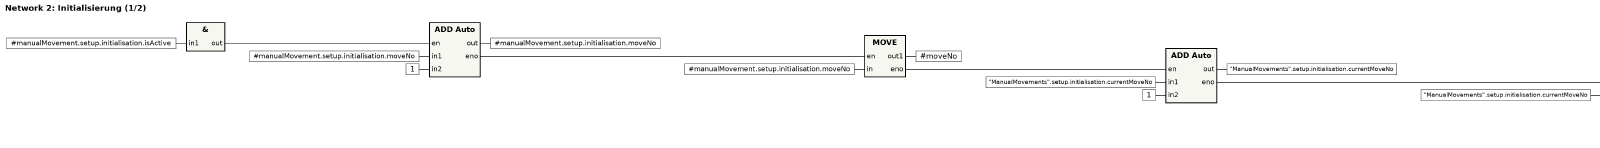
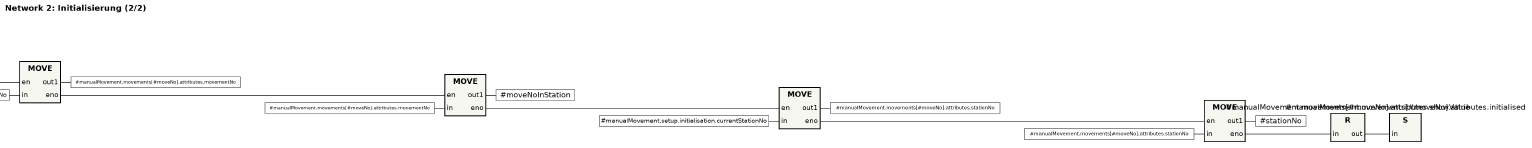
   IF #manualMovement.setup.initialisation.isActive THEN
       #manualMovement.setup.initialisation.moveNo := #manualMovement.setup.initialisation.moveNo + 1;
       #moveNo := #manualMovement.setup.initialisation.moveNo;
       "ManualMovements".setup.initialisation.currentMoveNo := "ManualMovements".setup.initialisation.currentMoveNo + 1;
       #manualMovement.movements[#moveNo].attributes.movementNo := "ManualMovements".setup.initialisation.currentMoveNo;
       #moveNoInStation := #manualMovement.movements[#moveNo].attributes.movementNo;
       #manualMovement.movements[#moveNo].attributes.stationNo := #manualMovement.setup.initialisation.currentStationNo;
       #stationNo := #manualMovement.movements[#moveNo].attributes.stationNo;
       #manualMovement.movements[#moveNo].attributes.showValue := FALSE;
       #manualMovement.movements[#moveNo].attributes.initialised := TRUE;
   END_IF;
END_REGION

REGION Network 3: Initialisierung abgeschlossen?
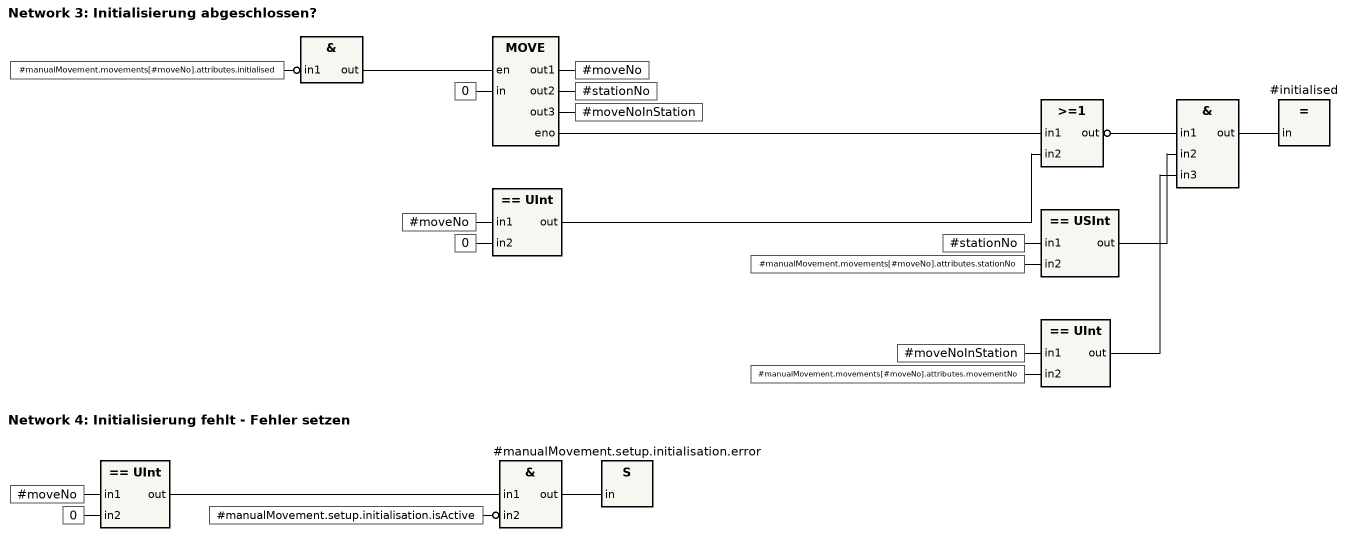
   #_w1 := NOT #manualMovement.movements[#moveNo].attributes.initialised;
   IF #_w1 THEN
       #moveNo := 0;
       #stationNo := 0;
       #moveNoInStation := 0;
   END_IF;
   #initialised := NOT (#_w1 OR (#moveNo = 0)) AND (#stationNo = #manualMovement.movements[#moveNo].attributes.stationNo) AND (#moveNoInStation = #manualMovement.movements[#moveNo].attributes.movementNo);
END_REGION

REGION Network 4: Initialisierung fehlt - Fehler setzen
   IF (#moveNo = 0) AND NOT #manualMovement.setup.initialisation.isActive THEN
       #manualMovement.setup.initialisation.error := TRUE;
   END_IF;
END_REGION

REGION Network 5: Sichtbarkeit
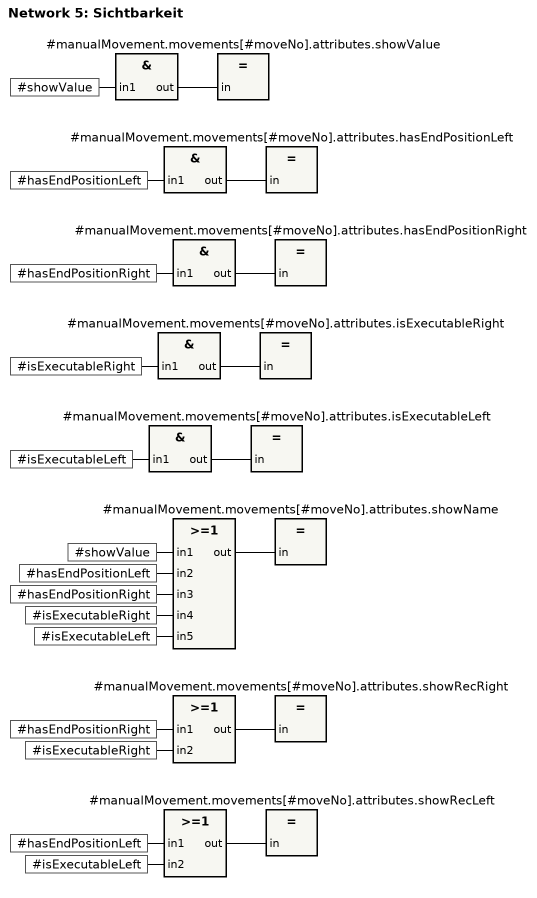
   #manualMovement.movements[#moveNo].attributes.showValue := #showValue;
   #manualMovement.movements[#moveNo].attributes.hasEndPositionLeft := #hasEndPositionLeft;
   #manualMovement.movements[#moveNo].attributes.hasEndPositionRight := #hasEndPositionRight;
   #manualMovement.movements[#moveNo].attributes.isExecutableRight := #isExecutableRight;
   #manualMovement.movements[#moveNo].attributes.isExecutableLeft := #isExecutableLeft;
   #manualMovement.movements[#moveNo].attributes.showName := #showValue OR #hasEndPositionLeft OR #hasEndPositionRight OR #isExecutableRight OR #isExecutableLeft;
   #manualMovement.movements[#moveNo].attributes.showRecRight := #hasEndPositionRight OR #isExecutableRight;
   #manualMovement.movements[#moveNo].attributes.showRecLeft := #hasEndPositionLeft OR #isExecutableLeft;
END_REGION
END_FUNCTION

FUNCTION "InitManualMovements" : Void   // FC909, SCL
{ S7_Optimized_Access := 'TRUE' }
VERSION : 0.1
   VAR_IN_OUT
      movements : Array[0.."SYS_MANUALMOVEMENTS"] of "typeManualMove";
   END_VAR
   VAR_TEMP
      tempCounter : USInt;
   END_VAR
BEGIN
   // Ersteller: Andreas Fast Automation
   // E-Mail: automation@fast-andreas.de
   //
   // Projekt dient zu Demonstrationszwecken und frei genutzt werden.
   //
   // Bausteinbeschreibung:
   // 


   FOR #tempCounter := 0 TO "SYS_MANUALMOVEMENTS" DO
       // Initialise all manual movements
       #movements[#tempCounter].attributes.initialised := false;
       "ManualMovements".movements[#tempCounter].attributes.showValue := false;
       "ManualMovements".movements[#tempCounter].attributes.showName := false;
       "ManualMovements".movements[#tempCounter].attributes.showRecRight := false;
       "ManualMovements".movements[#tempCounter].attributes.showRecLeft := false;
       "ManualMovements".movements[#tempCounter].attributes.isExecutableRight := false;
       "ManualMovements".movements[#tempCounter].attributes.isExecutableLeft := false;
       "ManualMovements".movements[#tempCounter].attributes.hasEndPositionRight := false;
       "ManualMovements".movements[#tempCounter].attributes.hasEndPositionLeft := false;

       #movements[#tempCounter].attributes.stationNo := 0;
       #movements[#tempCounter].attributes.movementNo := 0;
   END_FOR;
END_FUNCTION

// folder: 9. Library/9.2 Actors

FUNCTION_BLOCK "Actor"   // FB9200, FBD
TITLE = Aktoransteuerung
{ S7_Optimized_Access := 'TRUE' }
VERSION : 0.1
// Ersteller: Andreas Fast Automation
// E-Mail: automation@fast-andreas.de
// 
// Projekt dient zu Demonstrationszwecken und frei genutzt werden.
// 
// Bausteinbeschreibung:
// Grundlegende Funktionssteuerung eines Aktors
   VAR_INPUT
      config : USInt;   // Konfiguration Endschalterabfrage (0 = keine, 1 nur GS, 2 = Nur AS, 3 = Beide)
      "one-sided" : Bool;   // Einseitige Ansteuerung (Nur Ansteuerung zur Arbeitsstellung vorhanden, tastend)
      selfLocking : Bool;   // 1 = Selbsthaltung aktiv (Steuerimpuls setzt das Ausgangssignal)
      selfLockingInSetup : Bool;   // 1 = Selbsthaltung nur im Einrichtbetrieb bei einseitiger Spule (Ausgangsansteuerung wird setzend im Einrichten)
      holdEndposition : Bool;   // 1 = hält Ausgangsansteuerung aufrecht, wenn Endposition erreicht wurde
      iniHomePos : Bool;   // Grundstellung erreicht
      iniWorkPos : Bool;   // Arbeitsstellung erreicht
      interlockHome : Bool := true;   // 1 = Ansteuerung Grundstellung freigegeben
      interlockWork : Bool := true;   // 1 = Ansteuerung Arbeitsstellung freigegeben
      reactionTime : Time := t#25ms;   // Endschalter Reaktionsverzögerung
      configNoReleaseCycle : Bool := false;   // 1 = Stationsfreigabe ist zur Ansteuerung nicht notwendig
   END_VAR
   VAR_OUTPUT
      manualMoveNo : UInt;   // Bewegungsnummer für Einrichtfunktion
      homePos : Bool;
      workPos : Bool;
   END_VAR
   VAR_IN_OUT
      actor : "typeActor";
      signals : "typeStationSignals";
      manualMovement : "typeManualMovements";
   END_VAR
   VAR
      statManualHomePos : Bool;
      statManualWorkPos : Bool;
      statSetHomeAct : Bool;
      statSetWorkAct : Bool;
      statActorManualMovement : "ActorManualMovement";
      instReactionHome : TON_TIME;
      instReactionWork : TON_TIME;
   END_VAR
   VAR_TEMP
      tempSelfLocking : Bool;
      tempHomePosConfig : Bool;
      tempWorkPosConfig : Bool;
   END_VAR
BEGIN

REGION Network 1: Selbsthaltung
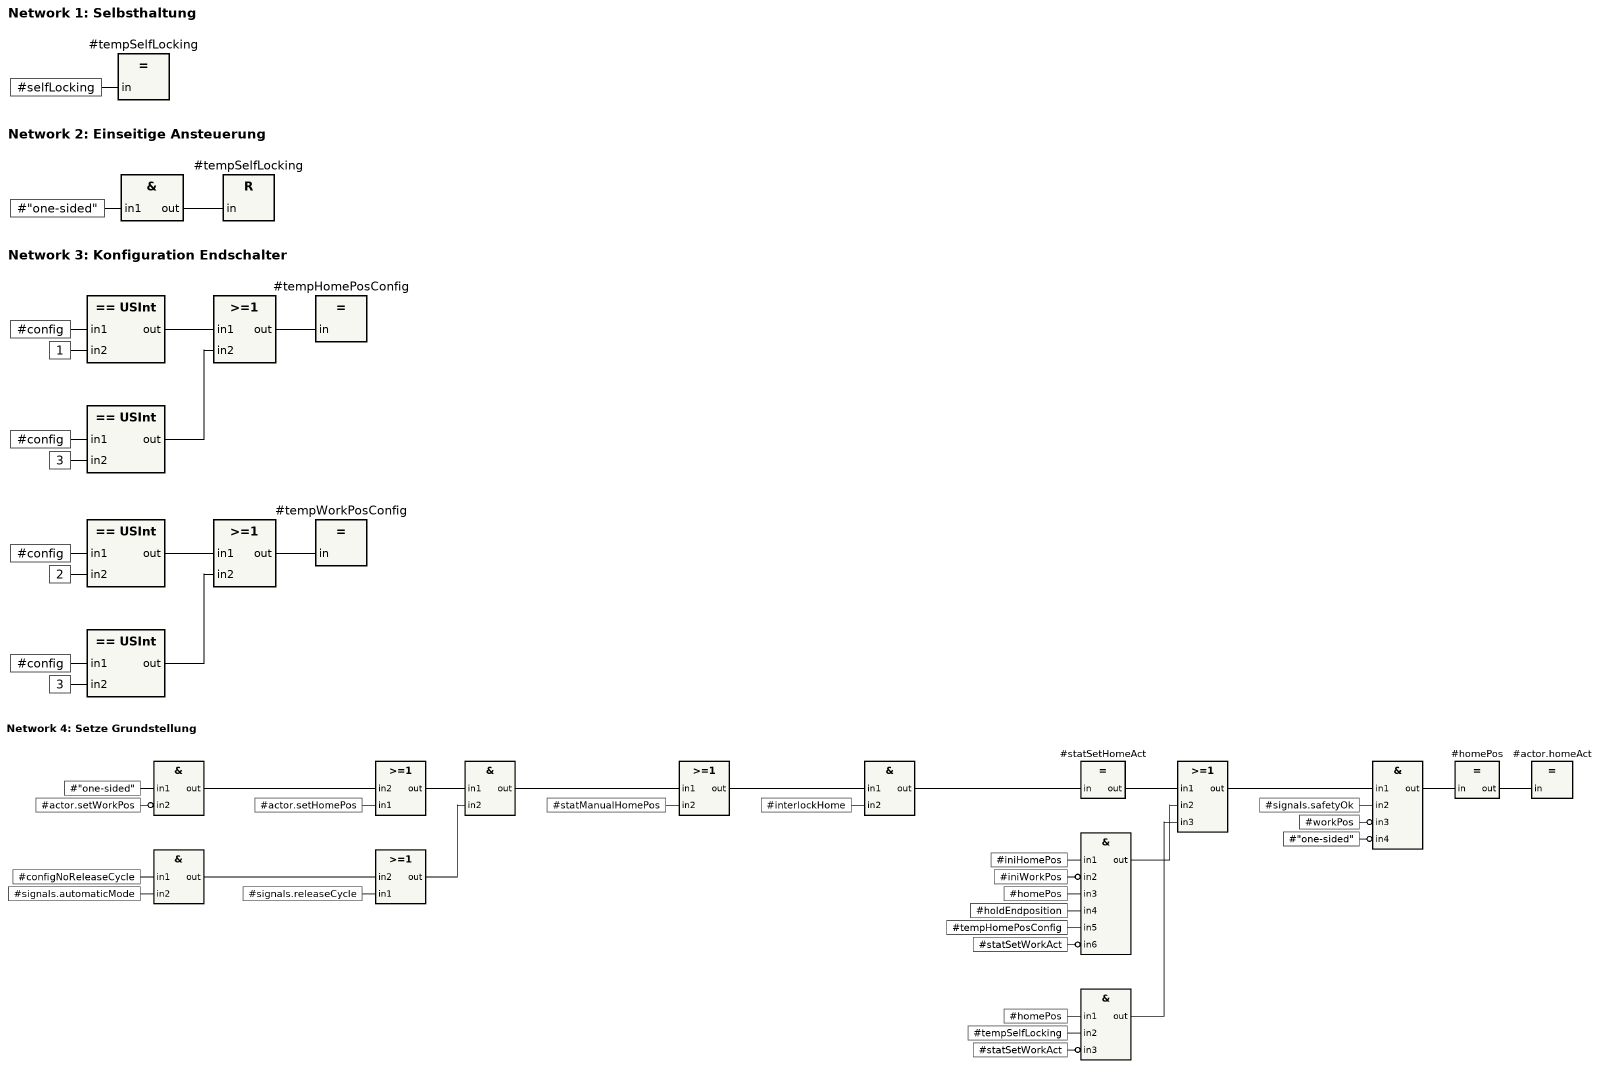
   #tempSelfLocking := #selfLocking;
END_REGION

REGION Network 2: Einseitige Ansteuerung
   IF #"one-sided" THEN #tempSelfLocking := FALSE; END_IF;
END_REGION

REGION Network 3: Konfiguration Endschalter
   // 0 = Ohne Inis
   // 1 = Nur Grundstellungsabfrage
   // 2 = Nur Arbeitstellungsabfrage
   // 3 = Beide Schaltstellungen werden abgefragt
   #tempHomePosConfig := (#config = 1) OR (#config = 3);
   #tempWorkPosConfig := (#config = 2) OR (#config = 3);
END_REGION

REGION Network 4: Setze Grundstellung
   #statSetHomeAct := ((((#"one-sided" AND NOT #actor.setWorkPos) OR #actor.setHomePos) AND ((#configNoReleaseCycle AND #signals.automaticMode) OR #signals.releaseCycle)) OR #statManualHomePos) AND #interlockHome;
   #homePos := (#statSetHomeAct OR (#iniHomePos AND NOT #iniWorkPos AND #homePos AND #holdEndposition AND #tempHomePosConfig AND NOT #statSetWorkAct) OR (#homePos AND #tempSelfLocking AND NOT #statSetWorkAct)) AND #signals.safetyOk AND NOT #workPos AND NOT #"one-sided";
   #actor.homeAct := #homePos;
END_REGION

REGION Network 5: Setze Arbeitsstellung
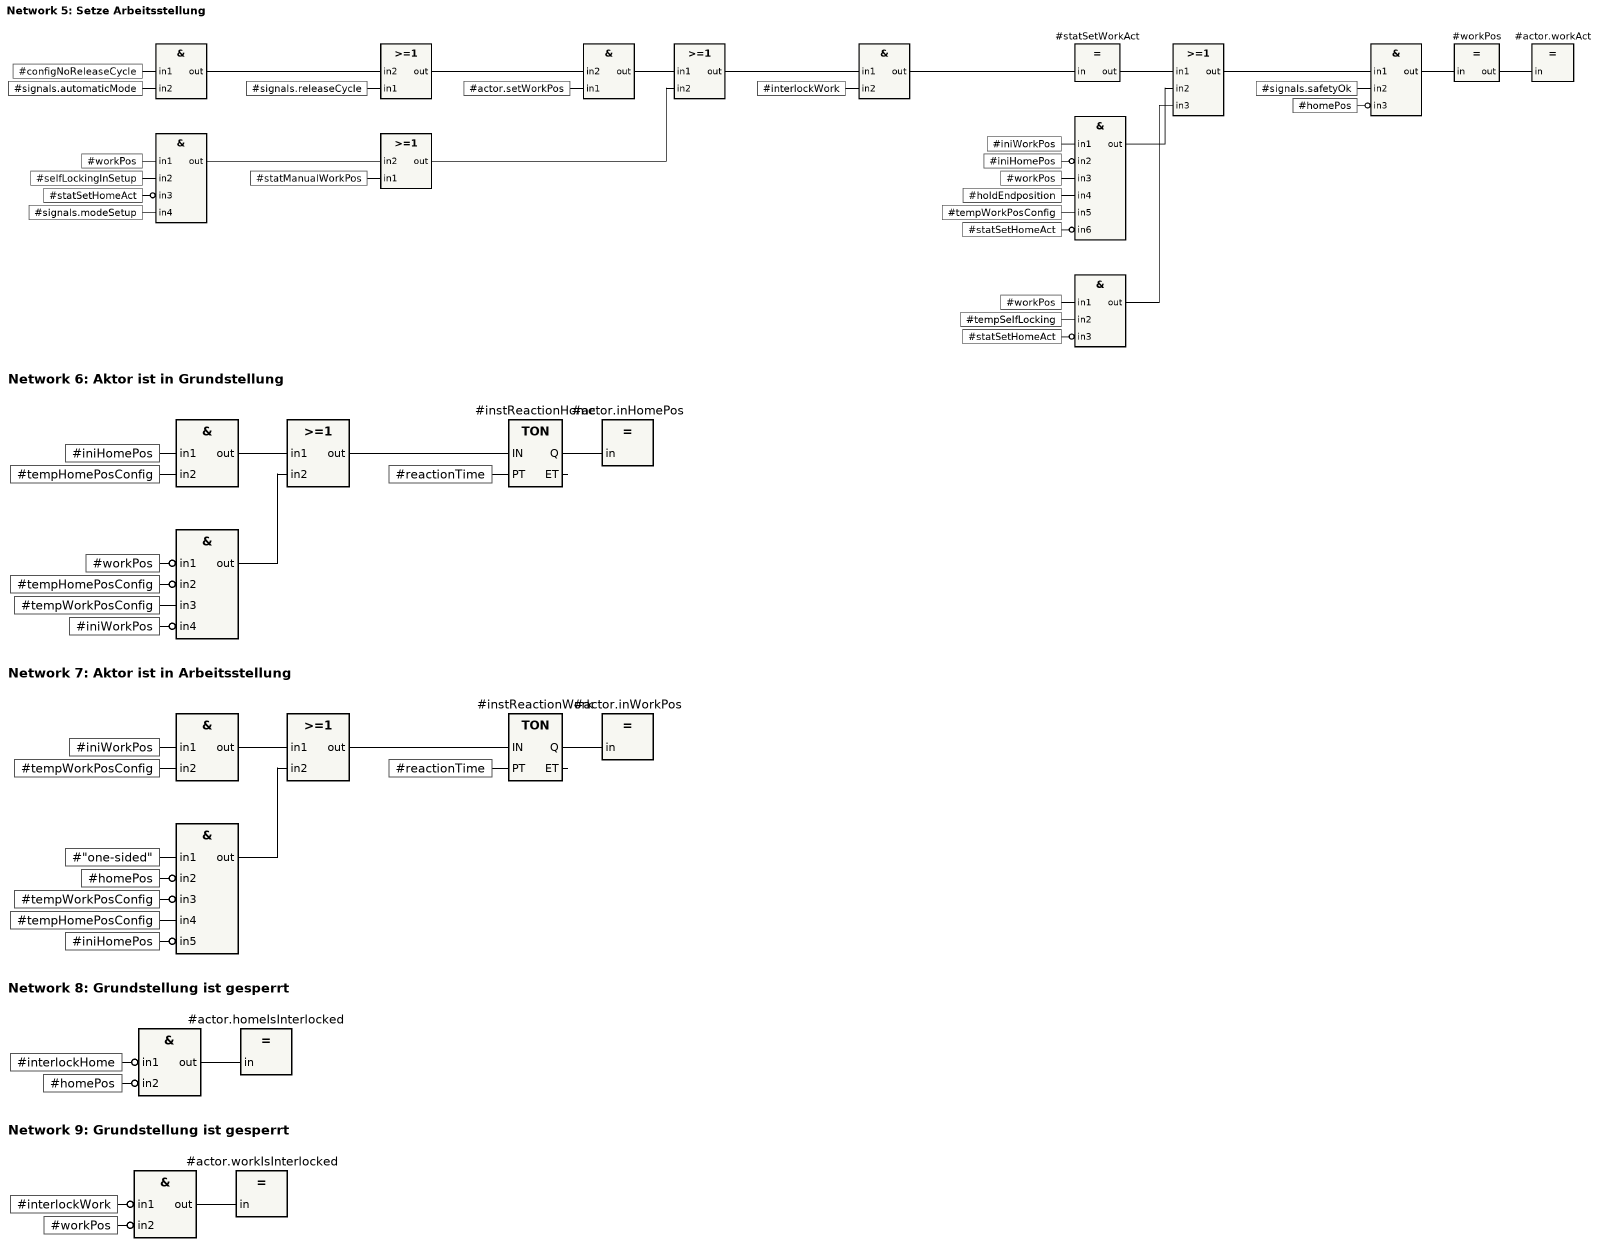
   #statSetWorkAct := ((((#configNoReleaseCycle AND #signals.automaticMode) OR #signals.releaseCycle) AND #actor.setWorkPos) OR (#workPos AND #selfLockingInSetup AND NOT #statSetHomeAct AND #signals.modeSetup) OR #statManualWorkPos) AND #interlockWork;
   #workPos := (#statSetWorkAct OR (#iniWorkPos AND NOT #iniHomePos AND #workPos AND #holdEndposition AND #tempWorkPosConfig AND NOT #statSetHomeAct) OR (#workPos AND #tempSelfLocking AND NOT #statSetHomeAct)) AND #signals.safetyOk AND NOT #homePos;
   #actor.workAct := #workPos;
END_REGION

REGION Network 6: Aktor ist in Grundstellung
   #instReactionHome(IN := (#iniHomePos AND #tempHomePosConfig) OR (NOT #workPos AND NOT #tempHomePosConfig AND #tempWorkPosConfig AND NOT #iniWorkPos),   // TON
                     PT := #reactionTime);
   #actor.inHomePos := #instReactionHome.Q;
END_REGION

REGION Network 7: Aktor ist in Arbeitsstellung
   #instReactionWork(IN := (#iniWorkPos AND #tempWorkPosConfig) OR (#"one-sided" AND NOT #homePos AND NOT #tempWorkPosConfig AND #tempHomePosConfig AND NOT #iniHomePos),   // TON
                     PT := #reactionTime);
   #actor.inWorkPos := #instReactionWork.Q;
END_REGION

REGION Network 8: Grundstellung ist gesperrt
   #actor.homeIsInterlocked := NOT #interlockHome AND NOT #homePos;
END_REGION

REGION Network 9: Grundstellung ist gesperrt
   #actor.workIsInterlocked := NOT #interlockWork AND NOT #workPos;
END_REGION

REGION Network 10: Steuerung Einrichtbewegung eines Aktors
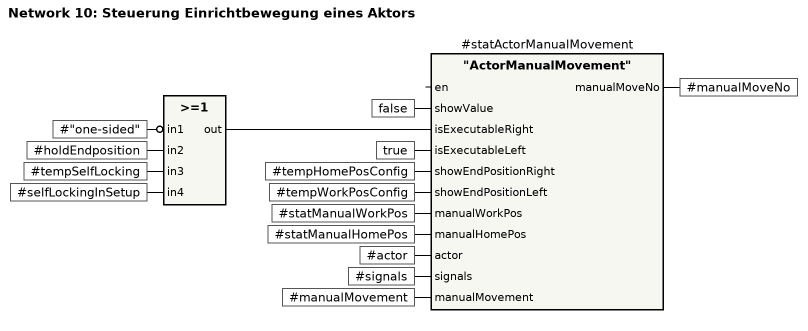
   #statActorManualMovement(showValue := false,   // "ActorManualMovement"
                           isExecutableRight := NOT #"one-sided" OR #holdEndposition OR #tempSelfLocking OR #selfLockingInSetup,
                           isExecutableLeft := true,
                           showEndPositionRight := #tempHomePosConfig,
                           showEndPositionLeft := #tempWorkPosConfig,
                           manualWorkPos := #statManualWorkPos,
                           manualHomePos := #statManualHomePos,
                           actor := #actor,
                           signals := #signals,
                           manualMovement := #manualMovement,
                           manualMoveNo => #manualMoveNo);
END_REGION
END_FUNCTION_BLOCK

FUNCTION_BLOCK "Actor_Reserved"   // FB9201, FBD
TITLE = Aktor als reservierter Platzhalter
{ S7_Optimized_Access := 'TRUE' }
VERSION : 0.1
// Ersteller: Andreas Fast Automation
// E-Mail: automation@fast-andreas.de
// 
// Projekt dient zu Demonstrationszwecken und frei genutzt werden.
// 
// Bausteinbeschreibung:
   VAR_OUTPUT
      manualMoveNo : UInt;   // Bewegungsnummer für Einrichtfunktion
   END_VAR
   VAR_IN_OUT
      manualMovement : "typeManualMovements";
   END_VAR
   VAR
      statActorManualMovement : "ActorManualMovement";
      sudtActor : "typeActor";
      sudtSignals : "typeStationSignals";
   END_VAR
BEGIN

REGION Network 1: Steuerung Einrichtbewegung eines Aktors
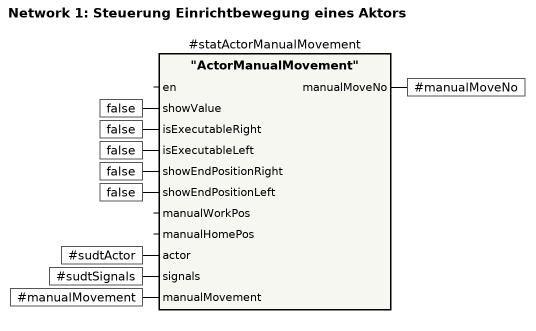
   #statActorManualMovement(showValue := false,   // "ActorManualMovement"
                           isExecutableRight := false,
                           isExecutableLeft := false,
                           showEndPositionRight := false,
                           showEndPositionLeft := false,
                           actor := #sudtActor,
                           signals := #sudtSignals,
                           manualMovement := #manualMovement,
                           manualMoveNo => #manualMoveNo);
END_REGION
END_FUNCTION_BLOCK

// folder: 9. Library/9.2 Actors/9.2.1 Cylinders

FUNCTION_BLOCK "Cylinder_2Out2In"   // FB9211, FBD
TITLE = Valve 2 Outs/2Ins
{ S7_Optimized_Access := 'TRUE' }
VERSION : 0.1
// Ersteller: Andreas Fast Automation
// E-Mail: automation@fast-andreas.de
// 
// Projekt dient zu Demonstrationszwecken und frei genutzt werden.
// 
// Bausteinbeschreibung:
// Ventilansteuerung
// Ansteuerung wird in AS/GS gehalten wenn zugehörige Endstellung vorhanden ist, selbst wenn die Aktoransteuerung rückgesetzt wird.
   VAR_INPUT
      iniHomePos : Bool;   // Grundstellung erreicht
      iniWorkPos : Bool;   // Arbeitsstellung erreicht
      interlockHome : Bool := true;   // 1 = Ansteuerung Grundstellung freigegeben
      interlockWork : Bool := true;   // 1 = Ansteuerung Arbeitsstellung freigegeben
      reactionTime : Time := t#25ms;   // Endschalter Reaktionsverzögerung
      monitoringTime : Time := T#10s;   // Überwachungszeit für Laufzeitfehler
      holdEndposition : Bool := true;   // 1 = hält Ausgangsansteuerung aufrecht, wenn Endposition erreicht wurde
   END_VAR
   VAR_OUTPUT
      manualMoveNo : UInt;   // Bewegungsnummer für Einrichtfunktion
      homePos : Bool;
      workPos : Bool;
   END_VAR
   VAR_IN_OUT
      actor : "typeActor_2Out2In";
      signals : "typeStationSignals";
      manualMovement : "typeManualMovements";
   END_VAR
   VAR
      instActor : "Actor";
      statActor : "typeActor";
      instMonitoringHome : TON_TIME;
      instMonitoringWork : TON_TIME;
   END_VAR
BEGIN

REGION Network 1: Verbinde Aktorsignale vor Aktoransteuerung
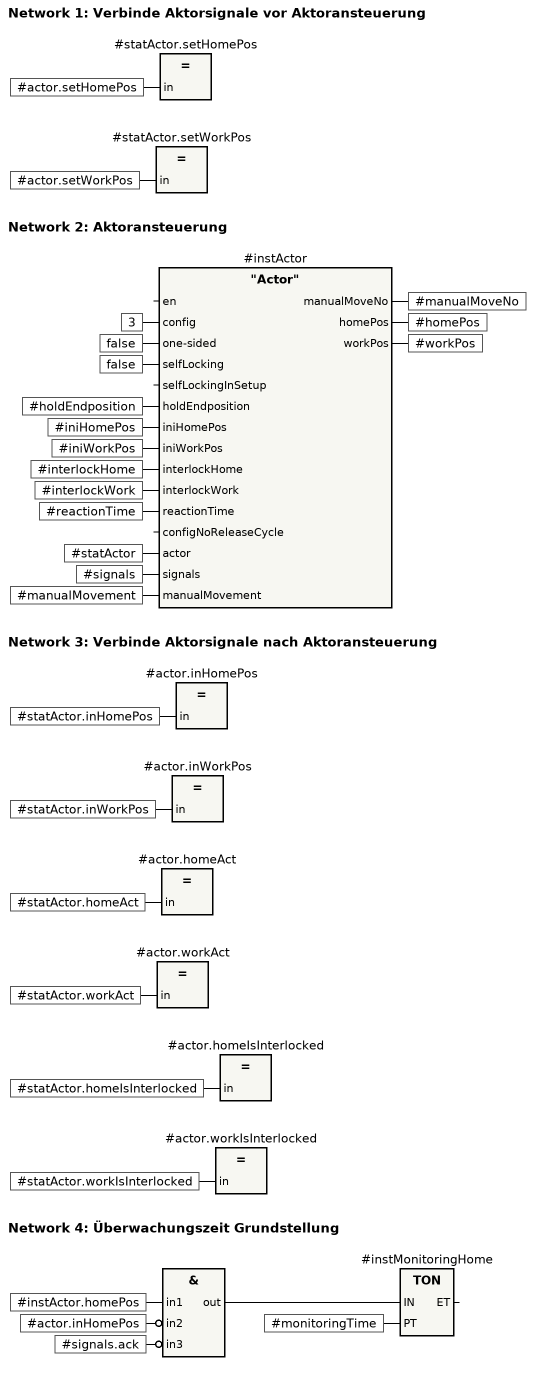
   #statActor.setHomePos := #actor.setHomePos;
   #statActor.setWorkPos := #actor.setWorkPos;
END_REGION

REGION Network 2: Aktoransteuerung
   #instActor(config := 3,   // "Actor"
              "one-sided" := false,
              selfLocking := false,
              holdEndposition := #holdEndposition,
              iniHomePos := #iniHomePos,
              iniWorkPos := #iniWorkPos,
              interlockHome := #interlockHome,
              interlockWork := #interlockWork,
              reactionTime := #reactionTime,
              actor := #statActor,
              signals := #signals,
              manualMovement := #manualMovement,
              manualMoveNo => #manualMoveNo,
              homePos => #homePos,
              workPos => #workPos);
END_REGION

REGION Network 3: Verbinde Aktorsignale nach Aktoransteuerung
   #actor.inHomePos := #statActor.inHomePos;
   #actor.inWorkPos := #statActor.inWorkPos;
   #actor.homeAct := #statActor.homeAct;
   #actor.workAct := #statActor.workAct;
   #actor.homeIsInterlocked := #statActor.homeIsInterlocked;
   #actor.workIsInterlocked := #statActor.workIsInterlocked;
END_REGION

REGION Network 4: Überwachungszeit Grundstellung
   #instMonitoringHome(IN := #instActor.homePos AND NOT #actor.inHomePos AND NOT #signals.ack,   // TON
                       PT := #monitoringTime);
END_REGION

REGION Network 5: Überwachungszeit Arbeitsstellung
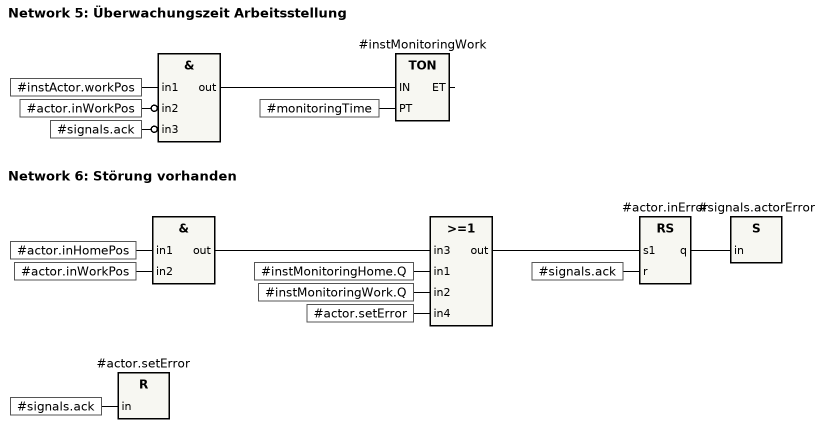
   #instMonitoringWork(IN := #instActor.workPos AND NOT #actor.inWorkPos AND NOT #signals.ack,   // TON
                       PT := #monitoringTime);
END_REGION

REGION Network 6: Störung vorhanden
   IF #signals.ack THEN
       #actor.inError := FALSE;   // RS flip-flop
   END_IF;
   IF (#actor.inHomePos AND #actor.inWorkPos) OR #instMonitoringHome.Q OR #instMonitoringWork.Q OR #actor.setError THEN
       #actor.inError := TRUE;
   END_IF;
   IF #actor.inError THEN #signals.actorError := TRUE; END_IF;
   IF #signals.ack THEN #actor.setError := FALSE; END_IF;
END_REGION
END_FUNCTION_BLOCK

FUNCTION_BLOCK "Cylinder_1Out2In"   // FB9212, FBD
TITLE = Valve 1 Outs/2Ins
{ S7_Optimized_Access := 'TRUE' }
VERSION : 0.1
// Ersteller: Andreas Fast Automation
// E-Mail: automation@fast-andreas.de
// 
// Projekt dient zu Demonstrationszwecken und frei genutzt werden.
// 
// Bausteinbeschreibung:
// Ventilansteuerung
// Ansteuerung wird in AS/GS gehalten wenn zugehörige Endstellung vorhanden ist, selbst wenn die Aktoransteuerung rückgesetzt wird.
   VAR_INPUT
      iniHomePos : Bool;   // Grundstellung erreicht
      iniWorkPos : Bool;   // Arbeitsstellung erreicht
      interlockWork : Bool := true;   // 1 = Ansteuerung Arbeitsstellung freigegeben
      reactionTime : Time := t#25ms;   // Endschalter Reaktionsverzögerung
      monitoringTime : Time := T#10s;   // Überwachungszeit für Laufzeitfehler
      holdEndposition : Bool := false;   // 1 = hält Ausgangsansteuerung aufrecht, wenn Endposition erreicht wurde
   END_VAR
   VAR_OUTPUT
      manualMoveNo : UInt;   // Bewegungsnummer für Einrichtfunktion
      workPos : Bool;   // SPS-Ausgang Ansteuerung Arbeitsstellung
   END_VAR
   VAR_IN_OUT
      actor : "typeActor_1Out2In";
      signals : "typeStationSignals";
      manualMovement : "typeManualMovements";
   END_VAR
   VAR
      instActor : "Actor";
      statActor : "typeActor";
      instMonitoringHome : TON_TIME;
      instMonitoringWork : TON_TIME;
   END_VAR
BEGIN

REGION Network 1: Verbinde Aktorsignale vor Aktoransteuerung
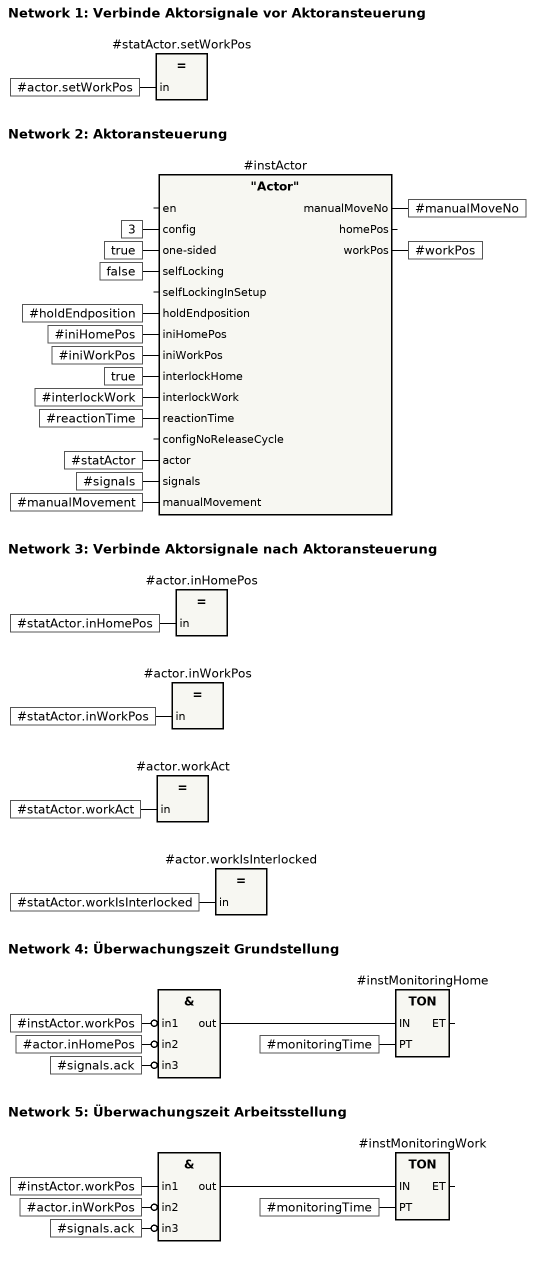
   #statActor.setWorkPos := #actor.setWorkPos;
END_REGION

REGION Network 2: Aktoransteuerung
   #instActor(config := 3,   // "Actor"
              "one-sided" := true,
              selfLocking := false,
              holdEndposition := #holdEndposition,
              iniHomePos := #iniHomePos,
              iniWorkPos := #iniWorkPos,
              interlockHome := true,
              interlockWork := #interlockWork,
              reactionTime := #reactionTime,
              actor := #statActor,
              signals := #signals,
              manualMovement := #manualMovement,
              manualMoveNo => #manualMoveNo,
              workPos => #workPos);
END_REGION

REGION Network 3: Verbinde Aktorsignale nach Aktoransteuerung
   #actor.inHomePos := #statActor.inHomePos;
   #actor.inWorkPos := #statActor.inWorkPos;
   #actor.workAct := #statActor.workAct;
   #actor.workIsInterlocked := #statActor.workIsInterlocked;
END_REGION

REGION Network 4: Überwachungszeit Grundstellung
   #instMonitoringHome(IN := NOT #instActor.workPos AND NOT #actor.inHomePos AND NOT #signals.ack,   // TON
                       PT := #monitoringTime);
END_REGION

REGION Network 5: Überwachungszeit Arbeitsstellung
   #instMonitoringWork(IN := #instActor.workPos AND NOT #actor.inWorkPos AND NOT #signals.ack,   // TON
                       PT := #monitoringTime);
END_REGION

REGION Network 6: Störung vorhanden
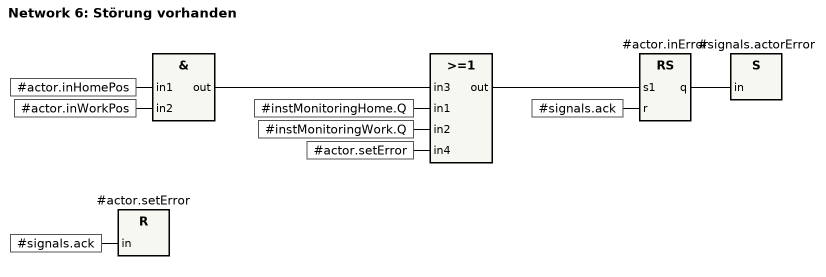
   IF #signals.ack THEN
       #actor.inError := FALSE;   // RS flip-flop
   END_IF;
   IF (#actor.inHomePos AND #actor.inWorkPos) OR #instMonitoringHome.Q OR #instMonitoringWork.Q OR #actor.setError THEN
       #actor.inError := TRUE;
   END_IF;
   IF #actor.inError THEN #signals.actorError := TRUE; END_IF;
   IF #signals.ack THEN #actor.setError := FALSE; END_IF;
END_REGION
END_FUNCTION_BLOCK

FUNCTION_BLOCK "Cylinder_2Out0In (ungetestet)"   // FB9213, FBD
TITLE = Valve 2 Outs/0Ins
{ S7_Optimized_Access := 'TRUE' }
VERSION : 0.1
// Ersteller: Andreas Fast Automation
// E-Mail: automation@fast-andreas.de
// 
// Projekt dient zu Demonstrationszwecken und frei genutzt werden.
// 
// Bausteinbeschreibung:
// Ventilansteuerung
// Ansteuerung wird in AS/GS gehalten wenn zugehörige Endstellung vorhanden ist, selbst wenn die Aktoransteuerung rückgesetzt wird.
   VAR_INPUT
      interlockHome : Bool := true;   // 1 = Ansteuerung Grundstellung freigegeben
      interlockWork : Bool := true;   // 1 = Ansteuerung Arbeitsstellung freigegeben
      reactionTime : Time := t#25ms;   // Endschalter Reaktionsverzögerung
   END_VAR
   VAR_OUTPUT
      manualMoveNo : UInt;   // Bewegungsnummer für Einrichtfunktion
      homePos : Bool;
      workPos : Bool;
   END_VAR
   VAR_IN_OUT
      actor : "typeActor_2Out0In";
      signals : "typeStationSignals";
      manualMovement : "typeManualMovements";
   END_VAR
   VAR
      instActor : "Actor";
      statActor : "typeActor";
   END_VAR
BEGIN

REGION Network 1: Verbinde Aktorsignale vor Aktoransteuerung
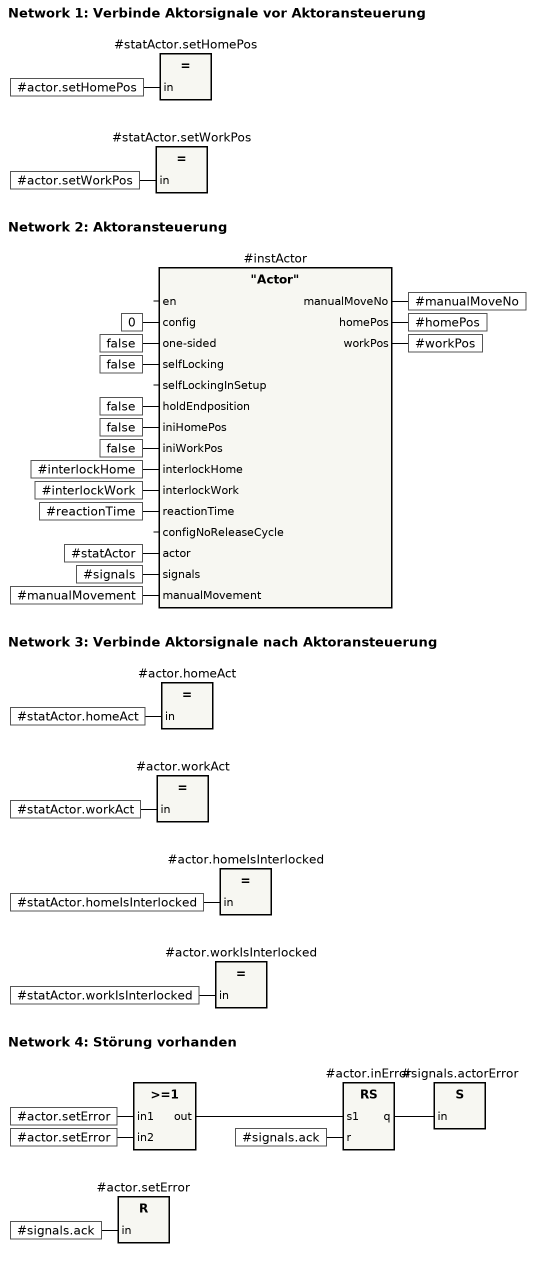
   #statActor.setHomePos := #actor.setHomePos;
   #statActor.setWorkPos := #actor.setWorkPos;
END_REGION

REGION Network 2: Aktoransteuerung
   #instActor(config := 0,   // "Actor"
              "one-sided" := false,
              selfLocking := false,
              holdEndposition := false,
              iniHomePos := false,
              iniWorkPos := false,
              interlockHome := #interlockHome,
              interlockWork := #interlockWork,
              reactionTime := #reactionTime,
              actor := #statActor,
              signals := #signals,
              manualMovement := #manualMovement,
              manualMoveNo => #manualMoveNo,
              homePos => #homePos,
              workPos => #workPos);
END_REGION

REGION Network 3: Verbinde Aktorsignale nach Aktoransteuerung
   #actor.homeAct := #statActor.homeAct;
   #actor.workAct := #statActor.workAct;
   #actor.homeIsInterlocked := #statActor.homeIsInterlocked;
   #actor.workIsInterlocked := #statActor.workIsInterlocked;
END_REGION

REGION Network 4: Störung vorhanden
   IF #signals.ack THEN
       #actor.inError := FALSE;   // RS flip-flop
   END_IF;
   IF #actor.setError OR #actor.setError THEN #actor.inError := TRUE; END_IF;
   IF #actor.inError THEN #signals.actorError := TRUE; END_IF;
   IF #signals.ack THEN #actor.setError := FALSE; END_IF;
END_REGION
END_FUNCTION_BLOCK

FUNCTION_BLOCK "Cylinder_2Out1In (ungetestet)"   // FB9214, FBD
TITLE = Valve 2 Outs/1Ins
{ S7_Optimized_Access := 'TRUE' }
VERSION : 0.1
// Ersteller: Andreas Fast Automation
// E-Mail: automation@fast-andreas.de
// 
// Projekt dient zu Demonstrationszwecken und frei genutzt werden.
// 
// Bausteinbeschreibung:
// Ventilansteuerung
// Ansteuerung wird in AS/GS gehalten wenn zugehörige Endstellung vorhanden ist, selbst wenn die Aktoransteuerung rückgesetzt wird.
   VAR_INPUT
      config : Bool;   // 0 = Ini zeigt Grundstellung erreicht / 1 = Ini zeigt Arbeitsstellung erreicht
      iniEndPos : Bool;   // SPS-Eingang Endposition erreicht
      interlockHome : Bool := true;   // 1 = Ansteuerung Grundstellung freigegeben
      interlockWork : Bool := true;   // 1 = Ansteuerung Arbeitsstellung freigegeben
      reactionTime : Time := t#25ms;   // Endschalter Reaktionsverzögerung
      monitoringTime : Time := T#10s;   // Überwachungszeit für Laufzeitfehler
      holdEndposition : Bool := false;   // 1 = hält Ausgangsansteuerung aufrecht, wenn Endposition erreicht wurde
   END_VAR
   VAR_OUTPUT
      manualMoveNo : UInt;   // Bewegungsnummer für Einrichtfunktion
      homePos : Bool;   // SPS-Ausgang Ansteuerung Grundstellung
      workPos : Bool;   // SPS-Ausgang Ansteuerung Arbeitsstellung
   END_VAR
   VAR_IN_OUT
      actor : "typeActor_2Out1In";
      signals : "typeStationSignals";
      manualMovement : "typeManualMovements";
   END_VAR
   VAR
      instActor : "Actor";
      statActor : "typeActor";
      instMonitoringHome : TON_TIME;
      instMonitoringWork : TON_TIME;
   END_VAR
   VAR_TEMP
      tusiConfig : USInt;
      txInHomePos : Bool;
      txInWorkPos : Bool;
   END_VAR
BEGIN

REGION Network 1: Verbinde Aktorsignale vor Aktoransteuerung
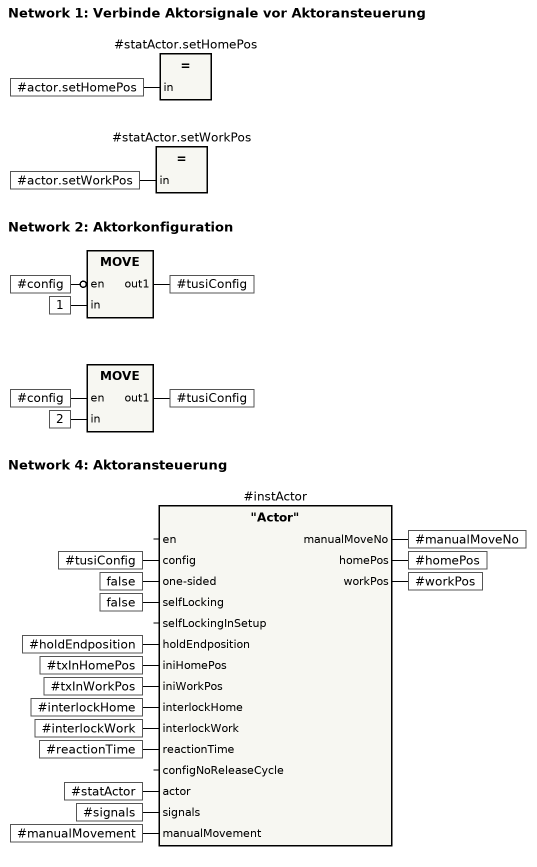
   #statActor.setHomePos := #actor.setHomePos;
   #statActor.setWorkPos := #actor.setWorkPos;
END_REGION

REGION Network 2: Aktorkonfiguration
   IF NOT #config THEN #tusiConfig := 1; END_IF;
   IF #config THEN #tusiConfig := 2; END_IF;
END_REGION

REGION Network 3 (SCL): Endschalter in Grundstellung/Arbeitsstellung

   IF NOT #config THEN // if sensor is checking home position
       #txInHomePos := #iniEndPos;
       #txInWorkPos := NOT #iniEndPos;

   ELSE // sensor is checking work position
       #txInWorkPos := #iniEndPos;
       #txInHomePos := NOT #iniEndPos;
   END_IF;
END_REGION

REGION Network 4: Aktoransteuerung
   #instActor(config := #tusiConfig,   // "Actor"
              "one-sided" := false,
              selfLocking := false,
              holdEndposition := #holdEndposition,
              iniHomePos := #txInHomePos,
              iniWorkPos := #txInWorkPos,
              interlockHome := #interlockHome,
              interlockWork := #interlockWork,
              reactionTime := #reactionTime,
              actor := #statActor,
              signals := #signals,
              manualMovement := #manualMovement,
              manualMoveNo => #manualMoveNo,
              homePos => #homePos,
              workPos => #workPos);
END_REGION

REGION Network 5: Verbinde Aktorsignale nach Aktoransteuerung
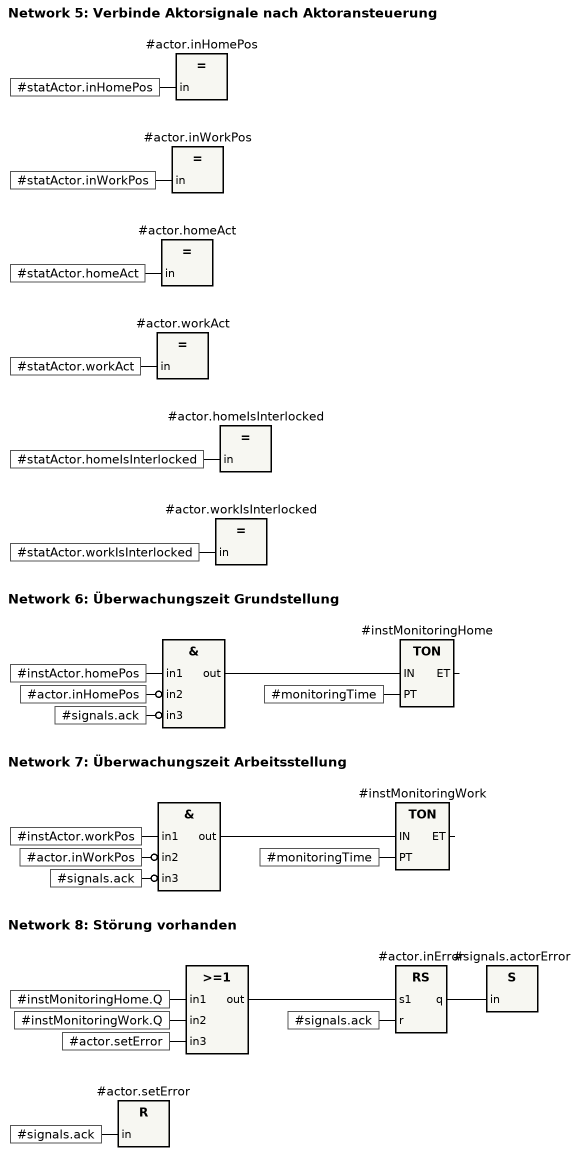
   #actor.inHomePos := #statActor.inHomePos;
   #actor.inWorkPos := #statActor.inWorkPos;
   #actor.homeAct := #statActor.homeAct;
   #actor.workAct := #statActor.workAct;
   #actor.homeIsInterlocked := #statActor.homeIsInterlocked;
   #actor.workIsInterlocked := #statActor.workIsInterlocked;
END_REGION

REGION Network 6: Überwachungszeit Grundstellung
   #instMonitoringHome(IN := #instActor.homePos AND NOT #actor.inHomePos AND NOT #signals.ack,   // TON
                       PT := #monitoringTime);
END_REGION

REGION Network 7: Überwachungszeit Arbeitsstellung
   #instMonitoringWork(IN := #instActor.workPos AND NOT #actor.inWorkPos AND NOT #signals.ack,   // TON
                       PT := #monitoringTime);
END_REGION

REGION Network 8: Störung vorhanden
   IF #signals.ack THEN
       #actor.inError := FALSE;   // RS flip-flop
   END_IF;
   IF #instMonitoringHome.Q OR #instMonitoringWork.Q OR #actor.setError THEN #actor.inError := TRUE; END_IF;
   IF #actor.inError THEN #signals.actorError := TRUE; END_IF;
   IF #signals.ack THEN #actor.setError := FALSE; END_IF;
END_REGION
END_FUNCTION_BLOCK

FUNCTION_BLOCK "Cylinder_1Out1In (ungetestet)"   // FB9215, FBD
TITLE = Valve 1 Out/1In
{ S7_Optimized_Access := 'TRUE' }
VERSION : 0.1
// Ersteller: Andreas Fast Automation
// E-Mail: automation@fast-andreas.de
// 
// Projekt dient zu Demonstrationszwecken und frei genutzt werden.
// 
// Bausteinbeschreibung:
// Ventilansteuerung
// Ansteuerung wird in AS/GS gehalten wenn zugehörige Endstellung vorhanden ist, selbst wenn die Aktoransteuerung rückgesetzt wird.
   VAR_INPUT
      config : Bool;   // 0 = Ini zeigt Grundstellung erreicht / 1 = Ini zeigt Arbeitsstellung erreicht
      iniEndPos : Bool;   // SPS-Eingang Endposition erreicht
      interlockWork : Bool := true;   // 1 = Ansteuerung Arbeitsstellung freigegeben
      reactionTime : Time := t#25ms;   // Endschalter Reaktionsverzögerung
      monitoringTime : Time := T#10s;   // Überwachungszeit für Laufzeitfehler
      holdEndposition : Bool := false;   // 1 = hält Ausgangsansteuerung aufrecht, wenn Endposition erreicht wurde
      selfLockingInSetup : Bool;   // 1 = Selbsthaltung nur im Einrichtbetrieb (zweiseitige Ausgangsansteuerung setzend)
   END_VAR
   VAR_OUTPUT
      manualMoveNo : UInt;   // Bewegungsnummer für Einrichtfunktion
      workPos : Bool;   // SPS-Ausgang Ansteuerung Arbeitsstellung
   END_VAR
   VAR_IN_OUT
      actor : "typeActor_1Out1In";
      signals : "typeStationSignals";
      manualMovement : "typeManualMovements";
   END_VAR
   VAR
      instActor : "Actor";
      statActor : "typeActor";
      instMonitoringHome : TON_TIME;
      instMonitoringWork : TON_TIME;
   END_VAR
   VAR_TEMP
      tusiConfig : USInt;
      txInHomePos : Bool;
      txInWorkPos : Bool;
      txsetzendimeinrichten : Bool;
   END_VAR
BEGIN

REGION Network 1: Verbinde Aktorsignale vor Aktoransteuerung
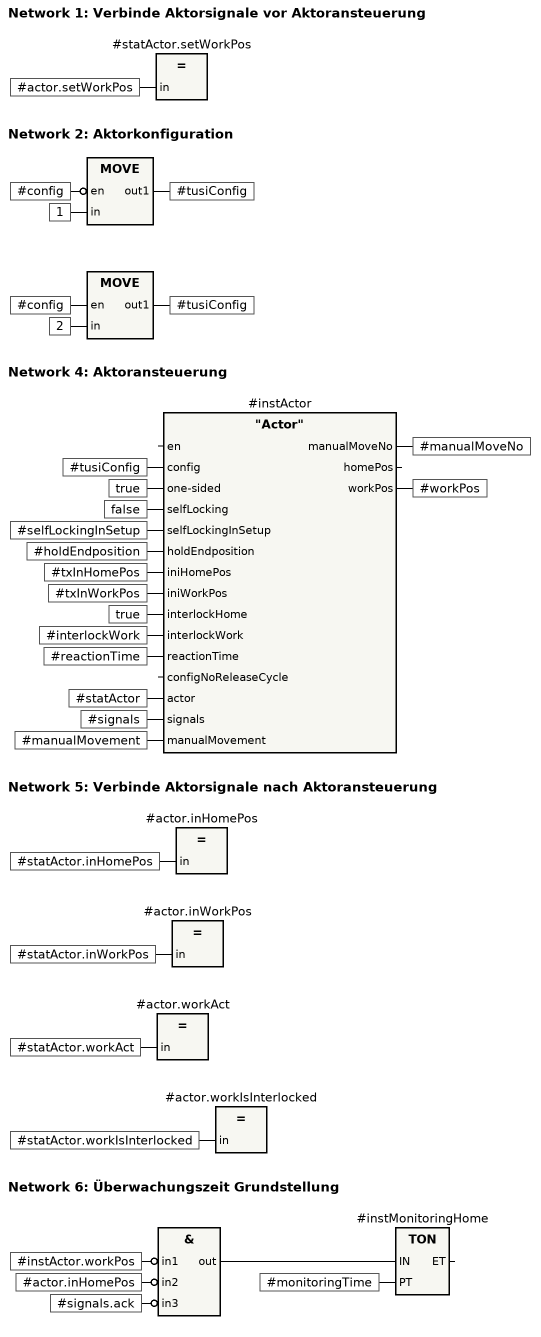
   #statActor.setWorkPos := #actor.setWorkPos;
END_REGION

REGION Network 2: Aktorkonfiguration
   IF NOT #config THEN #tusiConfig := 1; END_IF;
   IF #config THEN #tusiConfig := 2; END_IF;
END_REGION

REGION Network 3 (SCL): Endschalter in Grundstellung/Arbeitsstellung

   IF NOT #config THEN // if sensor is checking home position
       #txInHomePos := #iniEndPos;
       #txInWorkPos := NOT #iniEndPos;

   ELSE // sensor is checking work position
       #txInWorkPos := #iniEndPos;
       #txInHomePos := NOT #iniEndPos;
   END_IF;
END_REGION

REGION Network 4: Aktoransteuerung
   #instActor(config := #tusiConfig,   // "Actor"
              "one-sided" := true,
              selfLocking := false,
              selfLockingInSetup := #selfLockingInSetup,
              holdEndposition := #holdEndposition,
              iniHomePos := #txInHomePos,
              iniWorkPos := #txInWorkPos,
              interlockHome := true,
              interlockWork := #interlockWork,
              reactionTime := #reactionTime,
              actor := #statActor,
              signals := #signals,
              manualMovement := #manualMovement,
              manualMoveNo => #manualMoveNo,
              workPos => #workPos);
END_REGION

REGION Network 5: Verbinde Aktorsignale nach Aktoransteuerung
   #actor.inHomePos := #statActor.inHomePos;
   #actor.inWorkPos := #statActor.inWorkPos;
   #actor.workAct := #statActor.workAct;
   #actor.workIsInterlocked := #statActor.workIsInterlocked;
END_REGION

REGION Network 6: Überwachungszeit Grundstellung
   #instMonitoringHome(IN := NOT #instActor.workPos AND NOT #actor.inHomePos AND NOT #signals.ack,   // TON
                       PT := #monitoringTime);
END_REGION

REGION Network 7: Überwachungszeit Arbeitsstellung
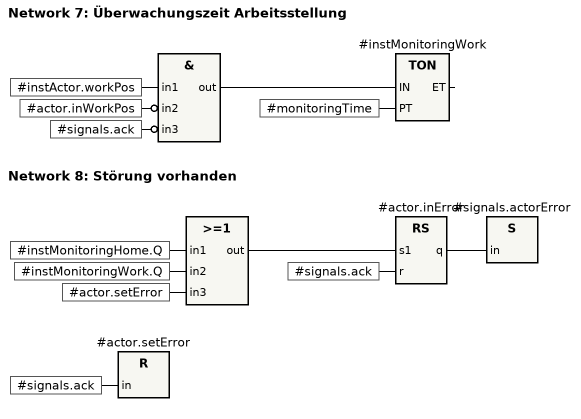
   #instMonitoringWork(IN := #instActor.workPos AND NOT #actor.inWorkPos AND NOT #signals.ack,   // TON
                       PT := #monitoringTime);
END_REGION

REGION Network 8: Störung vorhanden
   IF #signals.ack THEN
       #actor.inError := FALSE;   // RS flip-flop
   END_IF;
   IF #instMonitoringHome.Q OR #instMonitoringWork.Q OR #actor.setError THEN #actor.inError := TRUE; END_IF;
   IF #actor.inError THEN #signals.actorError := TRUE; END_IF;
   IF #signals.ack THEN #actor.setError := FALSE; END_IF;
END_REGION
END_FUNCTION_BLOCK

FUNCTION_BLOCK "Cylinder_1Out0In (ungetestet)"   // FB9216, FBD
TITLE = Valve 1 Out/0In
{ S7_Optimized_Access := 'TRUE' }
VERSION : 0.1
// Ersteller: Andreas Fast Automation
// E-Mail: automation@fast-andreas.de
// 
// Projekt dient zu Demonstrationszwecken und frei genutzt werden.
// 
// Bausteinbeschreibung:
// Ventilansteuerung
// Ansteuerung wird in AS/GS gehalten wenn zugehörige Endstellung vorhanden ist, selbst wenn die Aktoransteuerung rückgesetzt wird.
   VAR_INPUT
      interlockWork : Bool := true;   // 1 = Ansteuerung Arbeitsstellung freigegeben
      reactionTime : Time := t#25ms;   // Endschalter Reaktionsverzögerung
      holdEndposition : Bool := false;   // 1 = hält Ausgangsansteuerung aufrecht, wenn Endposition erreicht wurde
   END_VAR
   VAR_OUTPUT
      manualMoveNo : UInt;   // Bewegungsnummer für Einrichtfunktion
      workPos : Bool;   // SPS-Ausgang Ansteuerung Arbeitsstellung
   END_VAR
   VAR_IN_OUT
      actor : "typeActor_1Out0In";
      signals : "typeStationSignals";
      manualMovement : "typeManualMovements";
   END_VAR
   VAR
      instActor : "Actor";
      statActor : "typeActor";
   END_VAR
BEGIN

REGION Network 1: Verbinde Aktorsignale vor Aktoransteuerung
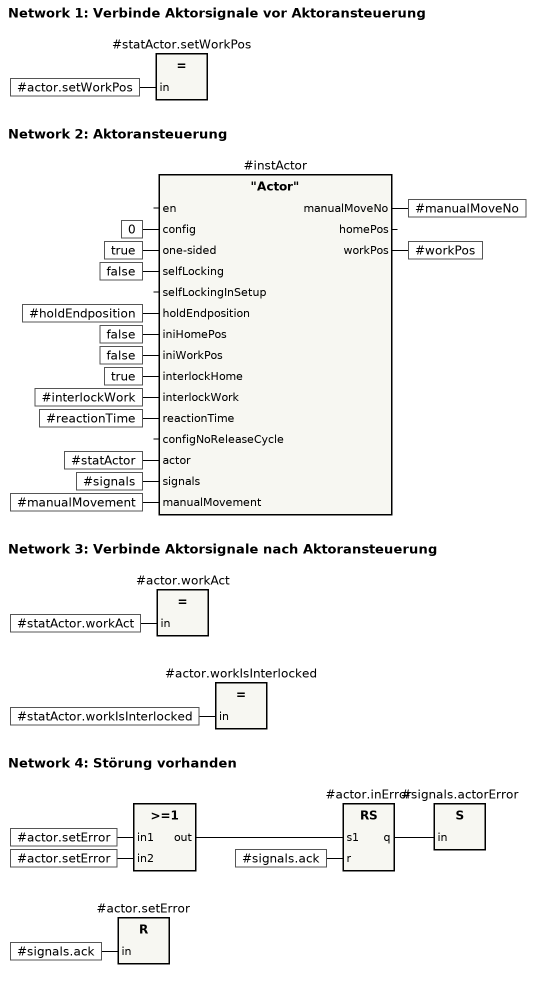
   #statActor.setWorkPos := #actor.setWorkPos;
END_REGION

REGION Network 2: Aktoransteuerung
   #instActor(config := 0,   // "Actor"
              "one-sided" := true,
              selfLocking := false,
              holdEndposition := #holdEndposition,
              iniHomePos := false,
              iniWorkPos := false,
              interlockHome := true,
              interlockWork := #interlockWork,
              reactionTime := #reactionTime,
              actor := #statActor,
              signals := #signals,
              manualMovement := #manualMovement,
              manualMoveNo => #manualMoveNo,
              workPos => #workPos);
END_REGION

REGION Network 3: Verbinde Aktorsignale nach Aktoransteuerung
   #actor.workAct := #statActor.workAct;
   #actor.workIsInterlocked := #statActor.workIsInterlocked;
END_REGION

REGION Network 4: Störung vorhanden
   IF #signals.ack THEN
       #actor.inError := FALSE;   // RS flip-flop
   END_IF;
   IF #actor.setError OR #actor.setError THEN #actor.inError := TRUE; END_IF;
   IF #actor.inError THEN #signals.actorError := TRUE; END_IF;
   IF #signals.ack THEN #actor.setError := FALSE; END_IF;
END_REGION
END_FUNCTION_BLOCK

// folder: 9. Library/9.2 Actors/9.2.2 Motors

FUNCTION_BLOCK "Motor_1Out"   // FB9221, FBD
TITLE = Motoransteuerung
{ S7_Optimized_Access := 'TRUE' }
VERSION : 0.1
// Ersteller: Andreas Fast Automation
// E-Mail: automation@fast-andreas.de
// 
// Projekt dient zu Demonstrationszwecken und frei genutzt werden.
// 
// Bausteinbeschreibung:
   VAR_INPUT
      circuitBreaker : Bool := true;   // 1 = Schutzschalter Ok
      interlockWork : Bool := true;   // 1 = Ansteuerung Arbeitsstellung freigegeben
      errorExtern : Bool;   // 1 = externer Fehler
   END_VAR
   VAR_OUTPUT
      manualMoveNo : UInt;   // Bewegungsnummer für Einrichtfunktion
      workPos : Bool;
   END_VAR
   VAR_IN_OUT
      actor : "typeActor_1Out0In";
      signals : "typeStationSignals";
      manualMovement : "typeManualMovements";
   END_VAR
   VAR
      instActor : "Actor";
      statActor : "typeActor";
   END_VAR
BEGIN

REGION Network 1: Verbinde Aktorsignale vor Aktoransteuerung
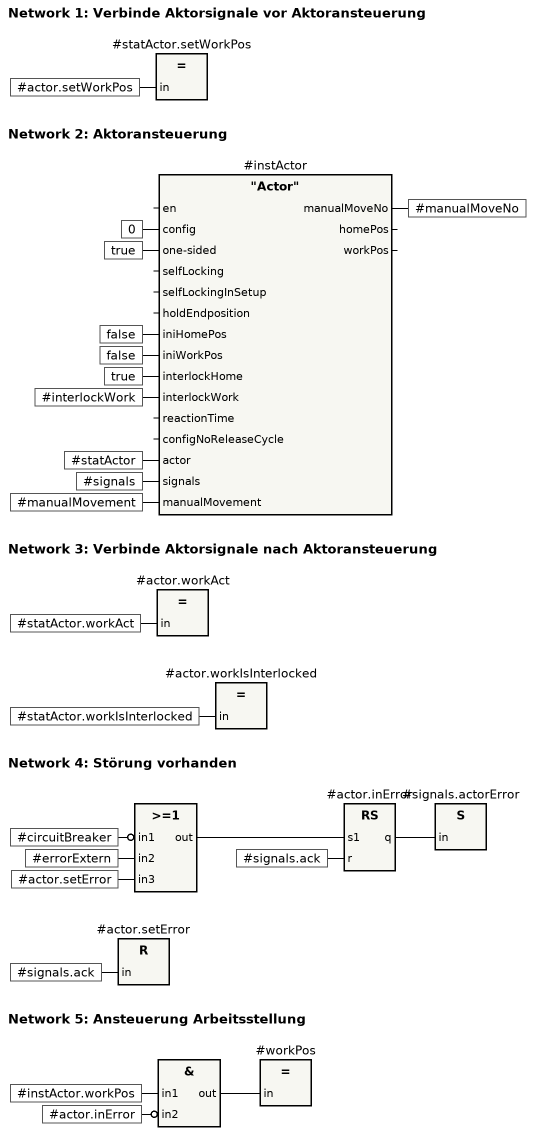
   #statActor.setWorkPos := #actor.setWorkPos;
END_REGION

REGION Network 2: Aktoransteuerung
   #instActor(config := 0,   // "Actor"
              "one-sided" := true,
              iniHomePos := false,
              iniWorkPos := false,
              interlockHome := true,
              interlockWork := #interlockWork,
              actor := #statActor,
              signals := #signals,
              manualMovement := #manualMovement,
              manualMoveNo => #manualMoveNo);
END_REGION

REGION Network 3: Verbinde Aktorsignale nach Aktoransteuerung
   #actor.workAct := #statActor.workAct;
   #actor.workIsInterlocked := #statActor.workIsInterlocked;
END_REGION

REGION Network 4: Störung vorhanden
   IF #signals.ack THEN
       #actor.inError := FALSE;   // RS flip-flop
   END_IF;
   IF NOT #circuitBreaker OR #errorExtern OR #actor.setError THEN #actor.inError := TRUE; END_IF;
   IF #actor.inError THEN #signals.actorError := TRUE; END_IF;
   IF #signals.ack THEN #actor.setError := FALSE; END_IF;
END_REGION

REGION Network 5: Ansteuerung Arbeitsstellung
   #workPos := #instActor.workPos AND NOT #actor.inError;
END_REGION
END_FUNCTION_BLOCK

FUNCTION_BLOCK "Motor_2Out"   // FB9222, FBD
TITLE = Motoransteuerung
{ S7_Optimized_Access := 'TRUE' }
VERSION : 0.1
// Ersteller: Andreas Fast Automation
// E-Mail: automation@fast-andreas.de
// 
// Projekt dient zu Demonstrationszwecken und frei genutzt werden.
// 
// Bausteinbeschreibung:
   VAR_INPUT
      circuitBreaker : Bool := true;   // 1 = Schutzschalter Ok
      interlockHome : Bool := true;   // 1 = Ansteuerung Grundstellung freigegeben
      interlockWork : Bool := true;   // 1 = Ansteuerung Arbeitsstellung freigegeben
      errorExtern : Bool;   // 1 = externer Fehler
      configNoReleaseCycle : Bool := false;   // 1 = Stationsfreigabe ist zur Ansteuerung nicht notwendig
   END_VAR
   VAR_OUTPUT
      manualMoveNo : UInt;   // Bewegungsnummer für Einrichtfunktion
      homePos : Bool;
      workPos : Bool;
   END_VAR
   VAR_IN_OUT
      actor : "typeActor_2Out0In";
      signals : "typeStationSignals";
      manualMovement : "typeManualMovements";
   END_VAR
   VAR
      instActor : "Actor";
      statActor : "typeActor";
   END_VAR
BEGIN

REGION Network 1: Verbinde Aktorsignale vor Aktoransteuerung
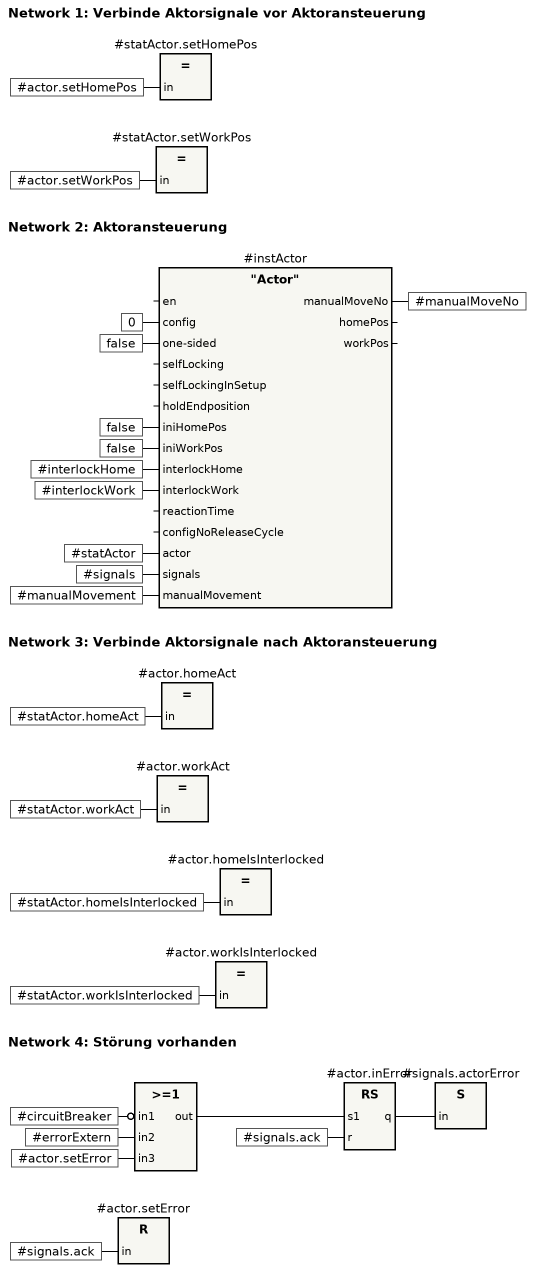
   #statActor.setHomePos := #actor.setHomePos;
   #statActor.setWorkPos := #actor.setWorkPos;
END_REGION

REGION Network 2: Aktoransteuerung
   #instActor(config := 0,   // "Actor"
              "one-sided" := false,
              iniHomePos := false,
              iniWorkPos := false,
              interlockHome := #interlockHome,
              interlockWork := #interlockWork,
              actor := #statActor,
              signals := #signals,
              manualMovement := #manualMovement,
              manualMoveNo => #manualMoveNo);
END_REGION

REGION Network 3: Verbinde Aktorsignale nach Aktoransteuerung
   #actor.homeAct := #statActor.homeAct;
   #actor.workAct := #statActor.workAct;
   #actor.homeIsInterlocked := #statActor.homeIsInterlocked;
   #actor.workIsInterlocked := #statActor.workIsInterlocked;
END_REGION

REGION Network 4: Störung vorhanden
   IF #signals.ack THEN
       #actor.inError := FALSE;   // RS flip-flop
   END_IF;
   IF NOT #circuitBreaker OR #errorExtern OR #actor.setError THEN #actor.inError := TRUE; END_IF;
   IF #actor.inError THEN #signals.actorError := TRUE; END_IF;
   IF #signals.ack THEN #actor.setError := FALSE; END_IF;
END_REGION

REGION Network 5: Ansteuerung Grundstellung
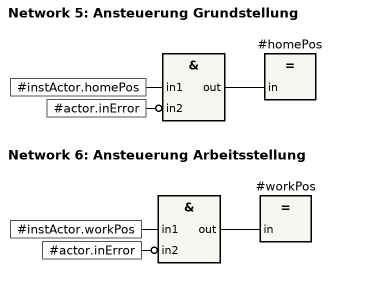
   #homePos := #instActor.homePos AND NOT #actor.inError;
END_REGION

REGION Network 6: Ansteuerung Arbeitsstellung
   #workPos := #instActor.workPos AND NOT #actor.inError;
END_REGION
END_FUNCTION_BLOCK

// folder: 9. Library/9.2 Actors/9.2.3 Drives

FUNCTION_BLOCK "Drive"   // FB9220, SCL
{ S7_Optimized_Access := 'TRUE' }
VERSION : 0.1
   VAR_INPUT
      minPosition : Real;   // minimale Position des Antriebs
      maxPosition : Real;   // maximale Position des Antriebs
      maxSpeed : Real;   // maximale Geschwindigkeit
      releasePos : Bool := true;   // 1 = Freigabe für positive Bewegung
      releaseNeg : Bool := true;   // 1 = Freigabe für negative Bewegung
      control : "typeDriveControl";   // Steuerbefehle
   END_VAR
   VAR_OUTPUT
      status : "typeDriveStatus";   // Status
   END_VAR
   VAR_IN_OUT
      setError : Bool;   // externer Fehler
      data : "typeDriveData";   // Einstelldaten
      converter : "typeDriveConverter";   // Drive <-> Umrichter
      signals : "typeStationSignals";   // Stationssignale
   END_VAR
   VAR
      statSetPositionLastCycle : Real;
      statNewPosition : Bool;
      statMoveToCommand : Bool;   // Fahrbefehl wurde aktiviert
      instTonJogMotion : TON_TIME;   // 1 = fortlaufende Bewegung
      instTrigJogPositiv : F_TRIG;
      instTrigJogNegativ : F_TRIG;
   END_VAR
   VAR_TEMP
      tempMoveCommandNumber : Int;
      tempInt : USInt;
      tempSetSpeed : Real;
      tempSetPosition : Real;   // Sollposition
      ValidMoveCommand : Bool;
   END_VAR
   // control.jog."step" := 5.0;
   // control.jog.speed := 1.0;
BEGIN
   // Ersteller: Andreas Fast Automation
   // E-Mail: automation@fast-andreas.de
   //
   // Projekt dient zu Demonstrationszwecken und frei genutzt werden.
   //
   // Bausteinbeschreibung:
   // 



   REGION Reset
       // Beim Reset alle anstehenden Fahrbefehle zurücksetzen
       IF #signals.resetCycle THEN
           FOR #tempInt := 1 TO "SYS_DRIVE_POSITIONS" DO
               #control.moveToPos[#tempInt] := false;
           END_FOR;
           #statMoveToCommand := false;
       END_IF;

   END_REGION



   REGION Automatic Mode
       //#statNewPosition := false;

       #tempMoveCommandNumber := "ReturnMoveCommand"(moveToPos := #control.moveToPos);
       #ValidMoveCommand := #tempMoveCommandNumber > 0;


   IF #signals.releaseCycle AND #ValidMoveCommand THEN // Ein Fahrbefehl ist vorhanden

       // Position des Fahrbefehls ansteuern
       #tempSetPosition := #data.position[#tempMoveCommandNumber];

       // Check position limits
       IF #tempSetPosition > #maxPosition THEN // limit end value positiv
           #tempSetPosition := #maxPosition;
       ELSIF #tempSetPosition < #minPosition THEN // limit end value negativ
           #tempSetPosition := #minPosition;
       END_IF;

       // check speed limit
       #tempSetSpeed := #data.speed[#tempMoveCommandNumber];
       IF #tempSetSpeed > #maxSpeed THEN
           #tempSetSpeed := #maxSpeed;
       END_IF;

       #converter.setPosition := #tempSetPosition;
       #converter.setSpeed := #tempSetSpeed;
       #statMoveToCommand := true;

   END_IF;

   END_REGION

   REGION Manual Mode

       IF #signals.modeSetup AND #signals.safetyOk THEN

           #instTrigJogPositiv(CLK := #control.jog.pos);
           #instTrigJogNegativ(CLK := #control.jog.neg);

           IF #instTrigJogPositiv.Q AND NOT #instTonJogMotion.Q THEN // Jump one step positiv
               IF #status.actualPosition + #control.jog.step > #maxPosition THEN
                   #tempSetPosition := #maxPosition;
               ELSE
                   #tempSetPosition := #status.actualPosition + #control.jog.step;
               END_IF;
               #converter.setPosition := #tempSetPosition;
               #statMoveToCommand := false;
           ELSIF #instTrigJogNegativ.Q AND NOT #instTonJogMotion.Q THEN // Jump one step negativ
               IF #status.actualPosition - #control.jog.step < #minPosition THEN
                   #tempSetPosition := #minPosition;
               ELSE
                   #tempSetPosition := #status.actualPosition - #control.jog.step;
               END_IF;
               #converter.setPosition := #tempSetPosition;
               #statMoveToCommand := false;
           ELSIF #control.jog.pos AND #instTonJogMotion.Q THEN // positiv continous motion 
               #converter.setPosition := #maxPosition;
               #statMoveToCommand := false;
           ELSIF #control.jog.neg AND #instTonJogMotion.Q THEN // negativ continous motion
               #converter.setPosition := #minPosition;
               #statMoveToCommand := false;
           ELSIF (#instTrigJogPositiv.Q XOR #instTrigJogNegativ.Q) AND #instTonJogMotion.Q THEN
               #converter.setPosition := #status.actualPosition; // stop at actual position when jogging is stopped
               #statMoveToCommand := false;
           END_IF;

           // Delay time for continous motion
           #instTonJogMotion(IN := #control.jog.pos XOR #control.jog.neg,
                             PT := t#1s);

           #converter.setSpeed := #control.jog.speed;

        END_IF;

   END_REGION

   REGION Stop On Current Position

       IF (NOT #ValidMoveCommand AND
           #signals.automaticMode) OR // Kein gültiger Fahrbefehl vorhanden
           NOT #signals.safetyOk OR
           #status.error OR
           (NOT #signals.modeSetup AND
           NOT #signals.automaticMode)
       THEN
           // Write actual position to set-position if drive has to stop
           #converter.setPosition := #status.actualPosition;
           #converter.setSpeed := 0.0;
           #statMoveToCommand := false;
        END_IF;   

    END_REGION

    REGION Check New Set Position

        // Set new position
        IF #statSetPositionLastCycle <> #converter.setPosition THEN
            #statNewPosition := true;
        ELSE
            #statNewPosition := false;
        END_IF;
        #statSetPositionLastCycle := #converter.setPosition;
    END_REGION


   REGION Release Motion

       #converter.releaseMotion :=
       #releasePos AND #converter.setPosition + #converter.posOffset > #converter.actualPosition OR
       #releaseNeg AND #converter.setPosition - #converter.posOffset < #converter.actualPosition;

       #status.interlockMin := NOT #releaseNeg AND NOT #converter.releaseMotion;
       #status.interlockMax := NOT #releasePos AND NOT #converter.releaseMotion;

   END_REGION

   REGION Status   
       // Status aktualisieren
       // 

       IF #signals.ack THEN
           #status.error := false;
           #setError := false;
       END_IF;
       IF #converter.error OR #setError THEN
           #status.error := true;
       END_IF;

       // Aktorstörung ausgeben
       IF #status.error THEN
           #signals.actorError := true;
       END_IF;

       #status.actualPosition := #converter.actualPosition;
       #status.actualSpeed := #converter.actualSpeed;
       #status.ready := #converter.ready AND NOT #status.error;
       #status.posReached := #converter.posReached AND NOT #statNewPosition AND #statMoveToCommand;
       #status.endPosMin := #status.actualPosition <= (#minPosition + 0.1);
       #status.endPosMax := #status.actualPosition >= (#maxPosition - 0.1);
       #status.inHomePos := #status.actualPosition > #data.position[1] - 1.0 AND #status.actualPosition < #data.position[1] + 1.0;

   END_REGION

   REGION Converter Signals
       // Signalaustausch mit dem Umrichter
       #converter.minPosDrive := #minPosition;
       #converter.maxPosDrive := #maxPosition;
       #converter.maxSpeedDrive := #maxSpeed;

   END_REGION
END_FUNCTION_BLOCK

FUNCTION_BLOCK "ConverterSEW"   // FB9223, SCL
{ S7_Optimized_Access := 'TRUE' }
VERSION : 0.1
   VAR_INPUT
      hwID : Hw_SubModule;   // Hardwarekennung des Submodules / Hardware identification of submodule
      circuitBreaker : Bool := true;   // 1 = Schutzschalter Ok
      minPosition : DInt;   // Minimale Position des Antriebs (Inkremente)
      maxPosition : DInt;   // Maximale Position des Antriebs (Inkremente)
      maxSpeed : DInt;   // Maximale Geschwindigkeit des Antriebs (Inkremente)
      posWindow : DInt;   // Positionsfenster (Inkremente)
      enable : Bool;   // Freigabe/Leistungsfreischaltung
   END_VAR
   VAR_OUTPUT
      commOk : Bool;
   END_VAR
   VAR_IN_OUT
      converter : "typeDriveConverter";   // Drive <-> Umrichter
      signals : "typeStationSignals";   // Stationssignale
   END_VAR
   VAR
      pdIn : Struct   // Prozessdaten Eingänge / process data inputs
         bit_0_0 : Bool;   // IPOS referenced
         bit_0_1 : Bool;   // IPOS positioned
         bit_0_2 : Bool;   // Virtual terminal
         bit_0_3 : Bool;   // Virtual terminal
         bit_0_4 : Bool;   // Virtual terminal
         bit_0_5 : Bool;   // Virtual terminal
         bit_0_6 : Bool;   // Virtual terminal
         bit_0_7 : Bool;   // Virtual terminal
         ampEnabled : Bool;   // Endstufe freigegeben / Power amplifier enabled
         converterReady : Bool;   // Bereit / Converter ready
         bit_1_2 : Bool;   // PA-data enabled
         bit_1_3 : Bool;   // Actual integrator set
         bit_1_4 : Bool;   // Actual parameter set
         error : Bool;   // Fehler / Warnung / Error / Warning
         limitSwitchLh : Bool;   // Endschalter Links aktiv / Limit switch left active
         limitSwitchRh : Bool;   // Endschalter Rechts aktiv / Limit switch right active
         actPos : DInt;   // 32Bit Istposition / 32-bit actual position
         actSpeed : Int;   // 16Bit Istdrehzahl / 16-bit actual speed
         res8 : Int;   // 16-bit actual active current
         res10 : Int;   // Reserved
      END_STRUCT;
      pdOut : Struct   // Prozessdaten Ausgänge / process data outputs
         bit_0_0 : Bool;   // Virtual terminal
         bit_0_1 : Bool;   // Virtual terminal
         bit_0_2 : Bool;   // Virtual terminal
         bit_0_3 : Bool;   // Virtual terminal
         bit_0_4 : Bool;   // Virtual terminal
         bit_0_5 : Bool;   // Virtual terminal
         bit_0_6 : Bool;   // Virtual terminal
         bit_0_7 : Bool;   // Virtual terminal
         contrInhibit : Bool;   // Reglersperre / Inhibit controller
         bit_1_1 : Bool;   // Rapid stop
         enableStop : Bool;   // Freigabe / Halt / Enable / Stop
         bit_1_3 : Bool;   // Holding control
         bit_1_4 : Bool;   // Ramp switchover
         bit_1_5 : Bool;   // Parameter set switchover
         resetError : Bool;   // Quittierung Fehler / Reset error
         bit_1_7 : Bool;   // Reserved
         setPos : DInt;   // 32Bit Sollposition / 32-bit target position
         setSpeed : Int;   // 16Bit Solldrehzahl / 16-bit target speed
         res8 : Int;   // 16-bit current limiting
         res10 : Int;   // 16-bit accelerate / decelerate ramp
      END_STRUCT;
      instGetIo : GETIO;   // Eingangsparameter lesen / Read input parameter
      instSetIo : SETIO;   // Ausgangsparameter schreiben / Write output parameter
      statGetIoStatus : DWord;   // Status 'GetIO' / Error information 'GetIO'
      statSetIoStatus : DWord;   // Status 'SetIO' / Error information 'SetIO'
      statConvFactorPos : Real;   // Umwandlungsfaktor für Position
      statConvFactorSpeed : Real;   // Umwandlugnsfaktor für Geschwindigkeit
      instResetError : TP_TIME;
   END_VAR
   VAR_TEMP
      tempPosReached : Bool;
      tempControlInhibit : Bool;
   END_VAR
BEGIN
   // Ersteller: Andreas Fast Automation
   // E-Mail: automation@fast-andreas.de
   //
   // Projekt dient zu Demonstrationszwecken und frei genutzt werden.
   //
   // Bausteinbeschreibung:
   // 


   REGION Convert Factors
       #statConvFactorPos := DINT_TO_REAL(#maxPosition - #minPosition) / (#converter.maxPosDrive - #converter.minPosDrive);
       #statConvFactorSpeed := DINT_TO_REAL(#maxSpeed) / #converter.maxSpeedDrive;

   END_REGION



   REGION Read Signals   

           // Read signals from converter
          #instGetIo(ID := #hwID,
                      STATUS => #statGetIoStatus,
                      INPUTS := #pdIn);
   END_REGION



   REGION Control 

       #instResetError(IN := #pdIn.error AND #signals.ack,
                       PT := T#500ms);

       IF #signals.ack THEN
           #converter.error := false;
       END_IF;
       IF NOT #circuitBreaker OR #pdIn.error THEN
           #converter.error := true;
       END_IF;

       #tempControlInhibit := #enable AND #signals.controlOn AND #signals.safetyOk;
       #pdOut.contrInhibit := NOT #tempControlInhibit;
       #pdOut.enableStop := #tempControlInhibit AND #converter.releaseMotion AND NOT #instResetError.Q;

       #pdOut.resetError := #instResetError.Q;


       #pdOut.setPos := REAL_TO_DINT(#converter.setPosition * #statConvFactorPos);
       #pdOut.setSpeed := REAL_TO_INT(#converter.setSpeed * #statConvFactorSpeed);


       #converter.ready := NOT #pdOut.contrInhibit 
       AND #pdOut.enableStop
       AND #pdIn.ampEnabled
       AND #pdIn.converterReady
       AND NOT #converter.error
       AND NOT #pdIn.limitSwitchLh
       AND NOT #pdIn.limitSwitchRh;

       #converter.actualSpeed := #pdIn.actSpeed / #statConvFactorSpeed;
       #converter.actualPosition := DINT_TO_REAL(#pdIn.actPos) / #statConvFactorPos;

       IF #pdOut.setPos < #pdIn.actPos THEN
           #tempPosReached:= (#pdIn.actPos - #pdOut.setPos) < #posWindow;
       ELSE
           #tempPosReached := (#pdOut.setPos - #pdIn.actPos) < #posWindow;
       END_IF;
       #converter.posReached := #tempPosReached AND #converter.ready;

       #converter.posOffset := (DINT_TO_REAL(#posWindow) / #statConvFactorPos) * 2.0;


   END_REGION



   REGION Write Signals

           // Send Data to converter
          #instSetIo(ID := #hwID,
                     STATUS => #statSetIoStatus,
                     OUTPUTS := #pdOut);

   END_REGION


   // Communication to converter is Ok
   IF #statGetIoStatus = 0 AND #statSetIoStatus = 0 THEN
       #commOk := true;
   ELSE
       #commOk := false;
       #converter.ready := false;
       #converter.error := true;
   END_IF;
END_FUNCTION_BLOCK

// folder: 9. Library/9.2 Actors/9.2.3 Drives/Drive Functions

FUNCTION "ReturnMoveCommand" : Int   // FC9221, SCL
{ S7_Optimized_Access := 'TRUE' }
FAMILY : Drive
VERSION : 0.1
   VAR_INPUT
      moveToPos : Array[1.."SYS_DRIVE_POSITIONS"] of Bool;
   END_VAR
   VAR_TEMP
      tempInt : USInt;   // Schleifenzähler
      tempMoveNumber : Int;
   END_VAR
   // Ret_Val : Bitnummer des Fahrbefehls. 0 = kein Fahrbefehl vorhanden
BEGIN
   // Ersteller: Andreas Fast Automation
   // E-Mail: automation@fast-andreas.de
   //
   // Projekt dient zu Demonstrationszwecken und frei genutzt werden.
   //
   // Bausteinbeschreibung:
   // 


   #tempMoveNumber := 0;

   // Prüfen ob ein Fahrbefehl ausgeführt werden soll
   FOR #tempInt := 1 TO "SYS_DRIVE_POSITIONS" DO
       // Statement section FOR
       IF #moveToPos[#tempInt] THEN
           IF #tempMoveNumber > 0 THEN // Prüfen ob mehrfache Fahrbefehle anstehen
               // Keinen Fahrbefehl ausgeben und Bausteinbearbeitung abbrechen
               #tempMoveNumber := 0;
               #ReturnMoveCommand := 0;
               RETURN;
           ELSE // noch kein Fahrbefehl vorhanden
               #tempMoveNumber := #tempInt;
           END_IF;
       END_IF;

   END_FOR;

   #ReturnMoveCommand := #tempMoveNumber;
END_FUNCTION

// folder: 9. Library/9.2 Actors/9.2.4 Robots

FUNCTION_BLOCK "RobotKuka"   // FB9231, FBD
TITLE = Steuerung KUKA Roboter
{ S7_Optimized_Access := 'TRUE' }
VERSION : 0.1
// Ersteller: Andreas Fast Automation
// E-Mail: automation@fast-andreas.de
// 
// Projekt dient zu Demonstrationszwecken und frei genutzt werden.
// 
// Bausteinbeschreibung:
   VAR_INPUT
      hwID : Hw_SubModule;   // Hardwarekennung des Submodules / Hardware identification of submodule
      homing : Bool;   // Start Grundstellungsfahrt
      start : Bool;   // Starte Auftrag
      job : UInt;   // Auftragsnummer
   END_VAR
   VAR_OUTPUT
      ready : Bool;   // Bereit
      busy : Bool;   // Auftrag läuft
      error : Bool;   // Fehler
      autoExt : Bool;   // Auto Ext aktiv
      stopped : Bool;   // Roboter ist gestoppt
      home : Bool;   // steht in Grundstellung
   END_VAR
   VAR_IN_OUT
      signals : "typeStationSignals";
      signalsRobIn : Variant;   // Eingangssignale von Roboter / Input signals from robot
      signalsRobOut : Variant;   // Ausgangssignale an Roboter / Output signals to robot
   END_VAR
   VAR
      pdIn : Struct   // Prozessdaten Eingänge / process data inputs
         autoExt : Struct   // Auto Extern Signale / Auto external signals
            res1 : Bool;   // A1 - Reserve / A1 - KRC control ready ($RC_RDY1)
            res2 : Bool;   // A2 -Reserve / A2 - IR ready ($PERI_RDY)
            res3 : Bool;   // A3 - Reserve / A3 - interface active ($I_O_ACTCONF)
            res4 : Bool;   // A4 - Systemmeldungen liegen an ($STOP_MESS) / A4 - system messages present ($STOP_MESS)
            proAct : Bool;   // A5 - Programm aktiv ($PRO_ACT) / A5 - program active ($PRO_ACT)
            proMove : Bool;   // A6 - Programmbewegung aktiv ($PRO_MOVE) / A6 - program movement active ($PRO_MOVE)
            robStopped : Bool;   // A7 - Roboter nicht in Bewegung ($ROB_STOPPED) / A7 - robot not moving ($ROB_STOPPED)
            modeExt : Bool;   // A8 - Betriebsart Automatik Extern ($EXT) / A8 - automatic mode external ($EXT)
            progNo : Byte;   // A9-16 Rückmeldung Auftragsnummer / A9-16 feedback job number
            modeT1 : Bool;   // A17 - Betriebsart T1 ($T1) / A17 - operation mode T1 ($T1)
            modeT2 : Bool;   // A18 - Betriebsart T2 ($T2) / A18 - operation mode T2 ($T2)
            res19 : Bool;   // A19 - Betriebsart Automatik ($AUT) / A19 - operation mode automatic ($AUT)
            pgnoReq : Bool;   // A20 - Bereit für Auftrag ($PGNO_REQ) / A20 - ready for job ($PGNO_REQ)
            inHome : Bool;   // A21 - Roboter in Grundstellung ($HOME) / A21 - robot in home position ($HOME)
            homing : Bool;   // A22 - Grundstellungsfahrt aktiv / A22 - home position run active
            res23 : Bool;   // A23 - Reserve / A23 - error in program sequence ($ALARM_STOP)
            userSafe : Bool;   // A24 - Bedienerschutz geschlossen ($USER_SAF) / A24 - user protection closed ($USER_SAF)
            failNo : Byte;   // A25-32 - Fehlermelde Code an SPS / A25-32 - failure code to PLC
            inHome1 : Bool;   // A33 - Grundstellungsposition Home 1 ($IN_HOME1) / A33 - in home position 1 ($IN_HOME1)
            inHome2 : Bool;   // A34 - Grundstellungsposition Home 2 ($IN_HOME2) / A34 - in home position 2 ($IN_HOME2)
            inHome3 : Bool;   // A35 - Grundstellungsposition Home 3 ($IN_HOME3) / A35 - in home position 3 ($IN_HOME3)
            inHome4 : Bool;   // A36 - Grundstellungsposition Home 4 ($IN_HOME4) / A36 - in home position 4 ($IN_HOME4)
            inHome5 : Bool;   // A37 - Grundstellungsposition Home 5 ($IN_HOME5) / A37 - in home position 5 ($IN_HOME5)
            inStandBy : Bool;   // A38 - Roboter in Parkposition / A38 - robot in stand by position
            res39 : Bool;   // A39 - / A39 - reference run is requested ($MASTERINGTEST_REQ_INT)
            res40 : Bool;   // A40 - / A40 - monitoring time referencing timed out ($MASTERINGTEST_MONTIME)
            res41 : Bool;   // A41 - / A41 - reference run active ($MASTERINGTEST_WORK)
            res42 : Bool;   // A42 - / A42 - error at adjustment referencing ($MASTERINGTEST_OK)
            res43 : Bool;   // A43 - / A43 - reference button functional ($MASTERINGSWITCH_OK)
            res44 : Bool;   // A44 - / A44 - monitoring time is exceeded ($BRAKETEST_MONTIME)
            res45 : Bool;   // A45 - / A45 - brake test is requested ($BRAKETEST_REQ_INT)
            res46 : Bool;   // A46 - / A46 - brake test active ($BRAKETEST_WORK)
            res47 : Bool;   // A47 - / A47 - brake is defective ($BRAKES_OK)
            res48 : Bool;   // A48 - / A48 - brake has reached wear limit ($BRAKETEST_WARN)
         END_STRUCT;
         userSignals : Array[0..9] of Byte;   // Benutzerdefinierte Signale / User defined signals
      END_STRUCT;
      pdOut : Struct   // Prozessdaten Ausgänge / process data outputs
         autoExt : Struct   // Auto Extern Signale / Auto external signals
            res1 : Bool;   // E1 - Reserve / E1 - external start ($EXT_START)
            moveEnable : Bool;   // E2 - Fahrfreigabe ($MOVE_ENABLE) / E2 - move enable ($MOVE_ENABLE)
            res3 : Bool;   // E3 - Externe Quittierung ($CONF_MESS) / E3 - external acknowledgement ($CONF_MESS)
            res4 : Bool;   // E4 - Reserve / E4 - external drives off ($DRIVES_OFF)
            drivesOn : Bool;   // E5 - Extern Antriebe Ein ($DRIVES_ON) / E5 - external drives on ($DRIVES_ON)
            ioAct : Bool;   // E6 - Extern Automatik Anforderung ($I_O_ACT) / E6 - external automatic request ($I_O_ACT)
            res7 : Bool;   // E7 - Reserve / E7 - reserve
            res8 : Bool;   // E8 - Reserve / E8 - reserve
            progNo : Byte;   // E9-16 - Auftragsnummer / E9-16 - job number
            pgnoValid : Bool;   // E17 - Auftrag übernehmen ($PGNO_VALID) / E17 - accept job ($PGNO_VALID)
            res18 : Bool;   // E18 - Reserve / E18 - reserve
            res19 : Bool;   // E19 - Reserve / E19 - reserve
            res20 : Bool;   // E20 - Reserve / E20 - stop after cycle end
            irHome : Bool;   // E21 - Roboter in Grundstellung fahren / E21 - move robot to home position
            res22 : Bool;   // E22 - Reserve / E22 - reserve
            res23 : Bool;   // E23 - Reserve / E23 - reserve
            res24 : Bool;   // E24 - Reserve / E24 - reserve
            res25 : Bool;   // E25 - Reserve / E25 - EKS user bit1
            res26 : Bool;   // E26 - Reserve / E25 - EKS user bit2
            res27 : Bool;   // E27 - Reserve / E25 - EKS user bit3
            res28 : Bool;   // E28 - Reserve / E25 - EKS user bit4
            res29 : Bool;   // E29 - Reserve / E29 - EKS toggle bit
            res30 : Bool;   // E30 - Reserve / E30 - reserve
            res31 : Bool;   // E31 - Reserve / E31 - reserve
            res32 : Bool;   // E32 - Reserve / E32 - reserve
            res33 : Bool;   // E33 - Reserve / E33 - reserve
            res34 : Bool;   // E34 - Reserve / E34 - reserve
            res35 : Bool;   // E35 - Reserve / E35 - reserve
            res36 : Bool;   // E36 - Reserve / E36 - reserve
            res37 : Bool;   // E37 - Reserve / E37 - reserve
            res38 : Bool;   // E38 - Reserve / E38 - reserve
            res39 : Bool;   // E39 - Reserve / E39 - request reference run ($MASTERINGTEST_REQ_EXT)
            res40 : Bool;   // E40 - Reserve / E40 - brake test request ($BRAKETEST_REQ_EXT)
            res41_48 : Byte;   // E41-48 - Reserve / E41-48 - reserve
         END_STRUCT;
         userSignals : Array[0..9] of Byte;   // Benutzerdefinierte Signale / User defined signals
      END_STRUCT;
      instGETIO : GETIO;   // Prozessabbild lesen / Read process image
      instSETIO : SETIO;   // Prozessabbild schreiben / Write process image
      statHoming : Struct   // Grundstellungsfahrt / Home position run
         req : Bool;   // Grundstellungsfahrt angefordert / Homing requested
         start : Bool;   // Start Grundstellungsfahrt / Start drive to home position
         busy : Bool;   // Grundstellungsfahrt läuft / Homing active
         done : Bool;   // Grundstellungsfahrt beendet / Homing done
         instResetPulse : TP_TIME;   // Impulsdauer Roboter Reset / Pulse duration robot reset
      END_STRUCT;
      statJob : Struct   // Auftragsbearbeitung / Job processing
         start : Bool;   // Programm starten / Start program
         setProgNo : Bool;   // Programmnummer setzen / Set program number
         progAck : Bool;   // Programm von Roboter bestätigt / Program acknowledged by robot
         busy : Bool;   // Programm läuft / Program busy
         done : Bool;   // Programm beendet - Ablauf löschen / Program done - reset sequence
      END_STRUCT;
      instRobStopped : TON_TIME;   // Verzögerungszeit Roboter nicht in Bewegung
   END_VAR
   VAR_TEMP
      tempPos : DInt;
      tempRetVal : Word;
      tempActJob : UInt;   // Aktuelle Auftragsnummer / Actual job number
      tempSetJob : UInt;   // Auftragsnummer Vorgabe / Job number specification
      tempErrFltRob : Bool;   // Störung im Roboterprogramm / Fault in the robot program
      tempErrCode : UInt;   // Störungsnummer / Error code
   END_VAR
BEGIN

REGION Network 1: Peripherie einlesen / Read periphery
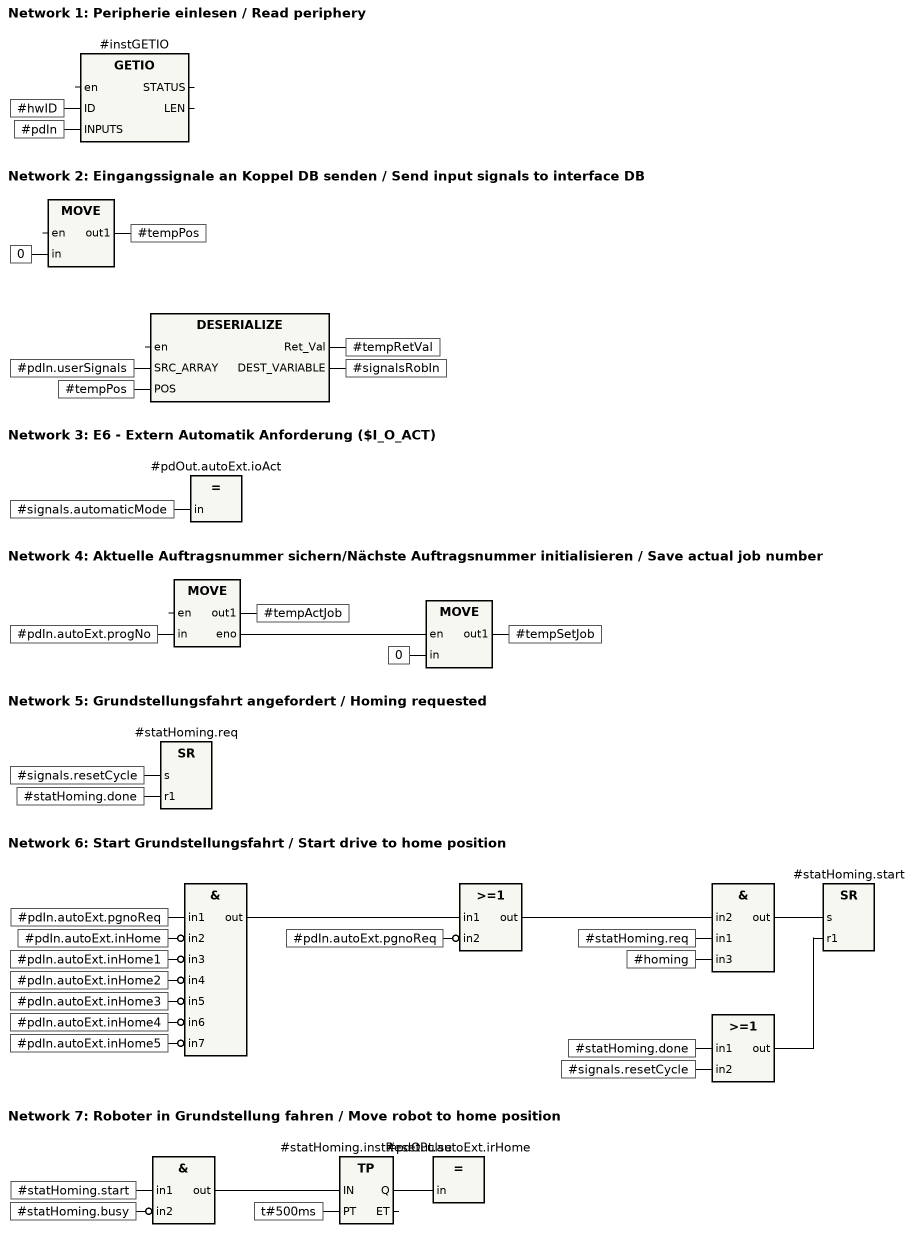
   #instGETIO(ID := #hwID, INPUTS := #pdIn);   // GETIO
END_REGION

REGION Network 2: Eingangssignale an Koppel DB senden / Send input signals to interface DB
   // no SCL statement known for Deserialize: written as a call
   #tempPos := 0;
   #tempRetVal := Deserialize(SRC_ARRAY := #pdIn.userSignals, POS := #tempPos, DEST_VARIABLE => #signalsRobIn);
END_REGION

REGION Network 3: E6 - Extern Automatik Anforderung ($I_O_ACT)
   #pdOut.autoExt.ioAct := #signals.automaticMode;
END_REGION

REGION Network 4: Aktuelle Auftragsnummer sichern/Nächste Auftragsnummer initialisieren / Save actual job number
   #tempActJob := #pdIn.autoExt.progNo;
   #tempSetJob := 0;
END_REGION

REGION Network 5: Grundstellungsfahrt angefordert / Homing requested
   IF #signals.resetCycle THEN
       #statHoming.req := TRUE;   // SR flip-flop
   END_IF;
   IF #statHoming.done THEN #statHoming.req := FALSE; END_IF;
END_REGION

REGION Network 6: Start Grundstellungsfahrt / Start drive to home position
   IF ((#pdIn.autoExt.pgnoReq AND NOT #pdIn.autoExt.inHome AND NOT #pdIn.autoExt.inHome1 AND NOT #pdIn.autoExt.inHome2 AND NOT #pdIn.autoExt.inHome3 AND NOT #pdIn.autoExt.inHome4 AND NOT #pdIn.autoExt.inHome5) OR NOT #pdIn.autoExt.pgnoReq) AND #statHoming.req AND #homing THEN
       #statHoming.start := TRUE;   // SR flip-flop
   END_IF;
   IF #statHoming.done OR #signals.resetCycle THEN #statHoming.start := FALSE; END_IF;
END_REGION

REGION Network 7: Roboter in Grundstellung fahren / Move robot to home position
   #statHoming.instResetPulse.TP(IN := #statHoming.start AND NOT #statHoming.busy, PT := t#500ms);
   #pdOut.autoExt.irHome := #statHoming.instResetPulse.Q;
END_REGION

REGION Network 8: Grundstellungsfahrt läuft / Homing active
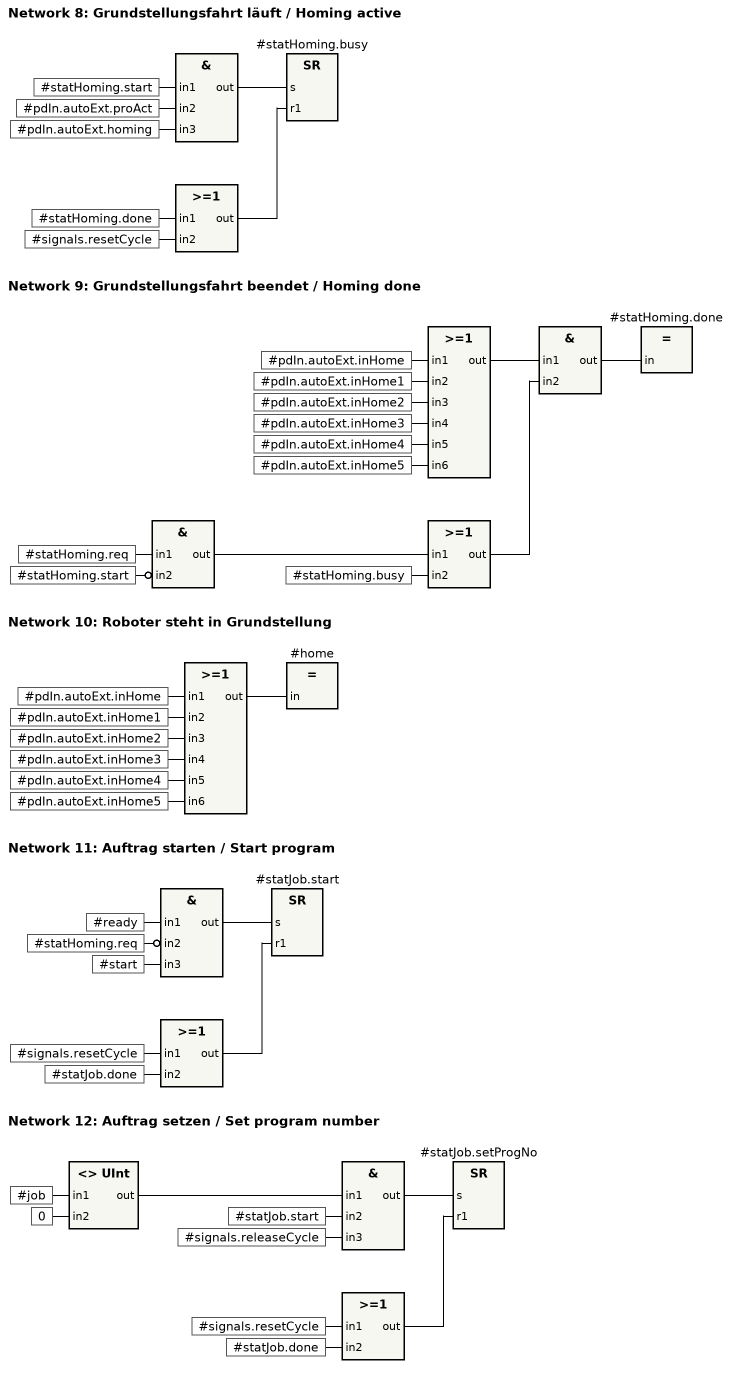
   IF #statHoming.start AND #pdIn.autoExt.proAct AND #pdIn.autoExt.homing THEN
       #statHoming.busy := TRUE;   // SR flip-flop
   END_IF;
   IF #statHoming.done OR #signals.resetCycle THEN #statHoming.busy := FALSE; END_IF;
END_REGION

REGION Network 9: Grundstellungsfahrt beendet / Homing done
   #statHoming.done := (#pdIn.autoExt.inHome OR #pdIn.autoExt.inHome1 OR #pdIn.autoExt.inHome2 OR #pdIn.autoExt.inHome3 OR #pdIn.autoExt.inHome4 OR #pdIn.autoExt.inHome5) AND ((#statHoming.req AND NOT #statHoming.start) OR #statHoming.busy);
END_REGION

REGION Network 10: Roboter steht in Grundstellung
   #home := #pdIn.autoExt.inHome OR #pdIn.autoExt.inHome1 OR #pdIn.autoExt.inHome2 OR #pdIn.autoExt.inHome3 OR #pdIn.autoExt.inHome4 OR #pdIn.autoExt.inHome5;
END_REGION

REGION Network 11: Auftrag starten / Start program
   IF #ready AND NOT #statHoming.req AND #start THEN
       #statJob.start := TRUE;   // SR flip-flop
   END_IF;
   IF #signals.resetCycle OR #statJob.done THEN #statJob.start := FALSE; END_IF;
END_REGION

REGION Network 12: Auftrag setzen / Set program number
   IF (#job <> 0) AND #statJob.start AND #signals.releaseCycle THEN
       #statJob.setProgNo := TRUE;   // SR flip-flop
   END_IF;
   IF #signals.resetCycle OR #statJob.done THEN #statJob.setProgNo := FALSE; END_IF;
END_REGION

REGION Network 13: Programmnummer vorgeben / Specify program number
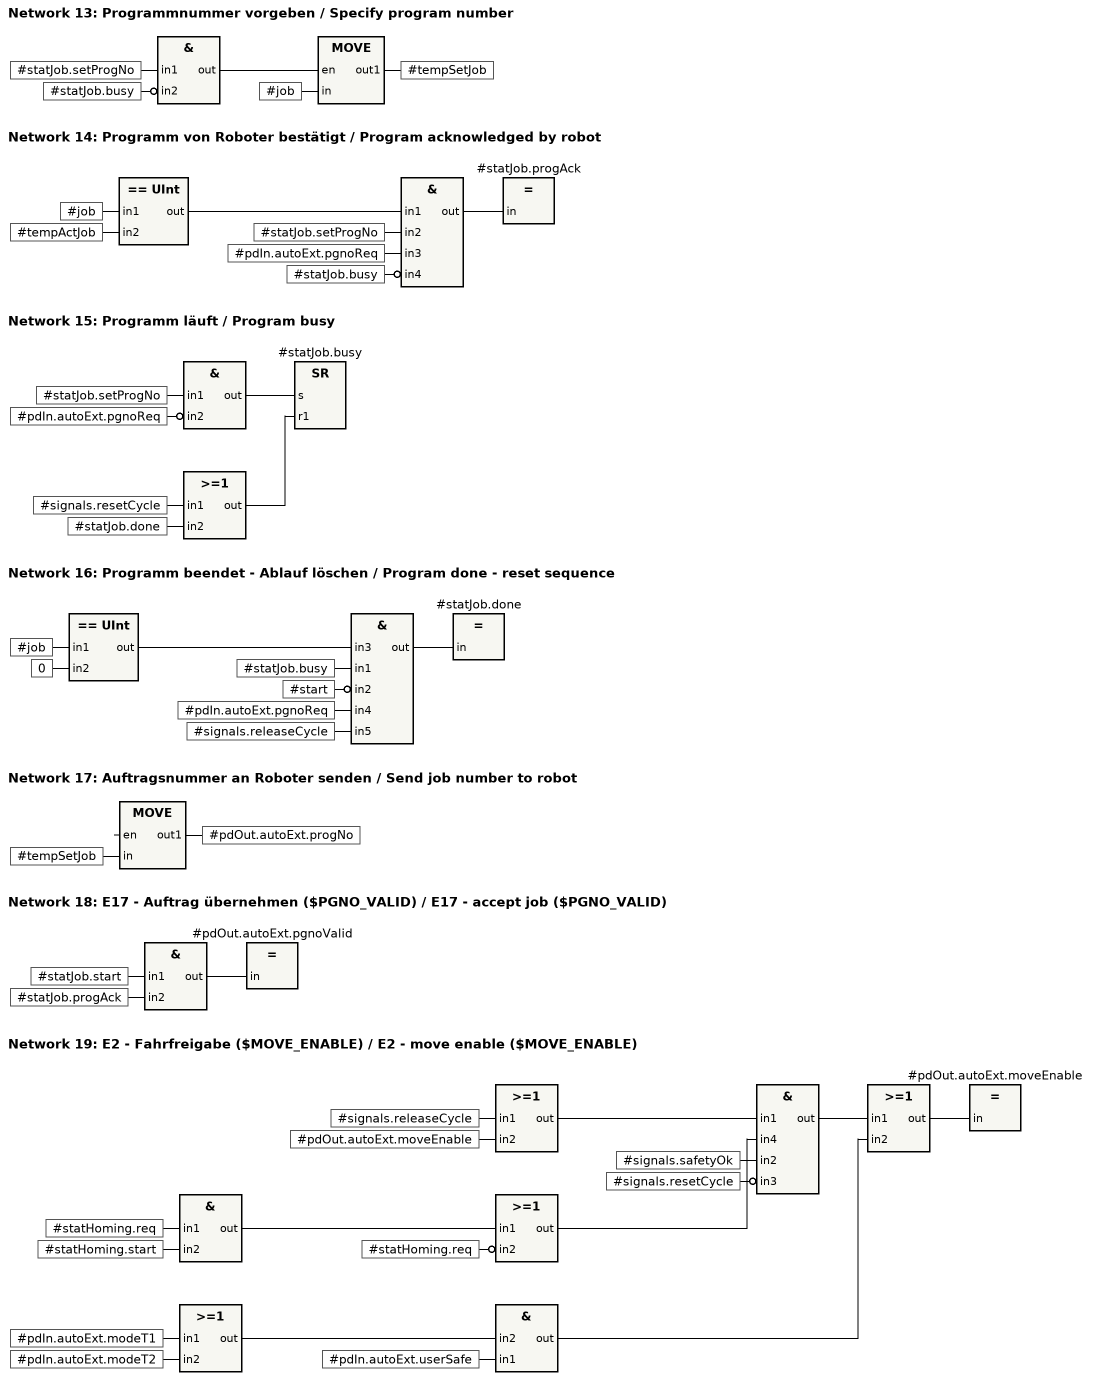
   IF #statJob.setProgNo AND NOT #statJob.busy THEN #tempSetJob := #job; END_IF;
END_REGION

REGION Network 14: Programm von Roboter bestätigt / Program acknowledged by robot
   #statJob.progAck := (#job = #tempActJob) AND #statJob.setProgNo AND #pdIn.autoExt.pgnoReq AND NOT #statJob.busy;
END_REGION

REGION Network 15: Programm läuft / Program busy
   IF #statJob.setProgNo AND NOT #pdIn.autoExt.pgnoReq THEN
       #statJob.busy := TRUE;   // SR flip-flop
   END_IF;
   IF #signals.resetCycle OR #statJob.done THEN #statJob.busy := FALSE; END_IF;
END_REGION

REGION Network 16: Programm beendet - Ablauf löschen / Program done - reset sequence
   #statJob.done := (#job = 0) AND #statJob.busy AND NOT #start AND #pdIn.autoExt.pgnoReq AND #signals.releaseCycle;
END_REGION

REGION Network 17: Auftragsnummer an Roboter senden / Send job number to robot
   #pdOut.autoExt.progNo := #tempSetJob;
END_REGION

REGION Network 18: E17 - Auftrag übernehmen ($PGNO_VALID) / E17 - accept job ($PGNO_VALID)
   #pdOut.autoExt.pgnoValid := #statJob.start AND #statJob.progAck;
END_REGION

REGION Network 19: E2 - Fahrfreigabe ($MOVE_ENABLE) / E2 - move enable ($MOVE_ENABLE)
   #pdOut.autoExt.moveEnable := ((#signals.releaseCycle OR #pdOut.autoExt.moveEnable) AND ((#statHoming.req AND #statHoming.start) OR NOT #statHoming.req) AND #signals.safetyOk AND NOT #signals.resetCycle) OR ((#pdIn.autoExt.modeT1 OR #pdIn.autoExt.modeT2) AND #pdIn.autoExt.userSafe);
END_REGION

REGION Network 20: Verzögerungszeit Roboter nicht in Bewegung
